SPLINE
SPL {X  -129.366, Y  +765.635, Z    +0.000, E1   +44.361, E3 -207865.968}
SPL {X  -144.719, Y  +739.715, Z    +0.000, E1   +37.620, E3 -207892.815}
SPL {X  -154.606, Y  +712.654, Z    +0.000, E1   +26.872, E3 -207906.035}
SPL {X  -158.229, Y  +695.175, Z    +0.000, E1   +17.621, E3 -207910.521}
SPL {X  -159.735, Y  +680.532, Z    +0.000, E1    +8.352, E3 -207912.613}
SPL {X  -159.976, Y  +673.579, Z    +0.000, E1    +3.308, E3 -207913.108}
SPL {X  -159.990, Y  +669.438, Z    +0.000, E1    +0.061, E3 -207913.205}
SPL {X  -159.990, Y  +667.221, Z    +0.000, E1    -2.789, E3 -207913.248}
SPL {X  -159.990, Y  +663.611, Z    +0.000, E1    -7.967, E3 -207913.439}
SPL {X  -159.990, Y  +658.381, Z    +0.000, E1   -16.786, E3 -207913.919}
SPL {X  -159.990, Y  +651.878, Z    +0.000, E1   -27.298, E3 -207914.918}
SPL {X  -159.990, Y  +644.587, Z    +0.000, E1   -37.284, E3 -207916.501}
SPL {X  -159.990, Y  +633.621, Z    +0.000, E1   -47.309, E3 -207919.992}
SPL {X  -159.990, Y  +588.658, Z    +0.000, E1   -60.812, E3 -207942.312}
SPL {X  -159.990, Y  +495.038, Z    +0.000, E1   -63.580, E3 -208017.548}
SPL {X  -159.990, Y  +483.848, Z    +0.000, E1   -63.590, E3 -208029.333}
SPL {X  -159.990, Y  +471.874, Z    +0.000, E1   -63.586, E3 -208041.959}
SPL {X  -159.990, Y  +461.079, Z    +0.000, E1   -63.579, E3 -208053.367}
SPL {X  -159.990, Y  +450.188, Z    +0.000, E1   -63.581, E3 -208064.858}
SPL {X  -159.990, Y  +442.553, Z    +0.000, E1   -63.337, E3 -208074.682}
ENDSPLINE

SPLINE
SPL {X  -159.990, Y  +465.419, Z    +0.000, E1   -58.181, E3 -208083.527}
ENDSPLINE

SPLINE
SPL {X  -159.990, Y  +455.003, Z    +0.000, E1   -58.788, E3 -208093.065}
SPL {X  -159.990, Y  +443.180, Z    +0.000, E1   -59.522, E3 -208103.103}
SPL {X  -159.990, Y  +431.227, Z    +0.000, E1   -60.120, E3 -208113.796}
SPL {X  -159.990, Y  +413.464, Z    +0.000, E1   -61.043, E3 -208128.786}
SPL {X  -159.990, Y  +395.417, Z    +0.000, E1   -62.063, E3 -208142.228}
SPL {X  -159.983, Y  +381.042, Z    +0.000, E1   -62.802, E3 -208152.860}
SPL {X  -159.542, Y  +370.537, Z    +0.000, E1   -63.069, E3 -208162.242}
SPL {X  -158.758, Y  +362.683, Z    +0.000, E1   -62.956, E3 -208171.515}
SPL {X  -157.125, Y  +352.357, Z    +0.000, E1   -62.751, E3 -208184.249}
SPL {X  -154.421, Y  +340.656, Z    +0.000, E1   -62.344, E3 -208199.602}
SPL {X  -151.938, Y  +332.383, Z    +0.000, E1   -61.927, E3 -208211.075}
SPL {X  -149.604, Y  +325.796, Z    +0.000, E1   -61.568, E3 -208220.461}
SPL {X  -147.413, Y  +320.320, Z    +0.000, E1   -61.198, E3 -208228.514}
SPL {X  -145.235, Y  +315.391, Z    +0.000, E1   -60.847, E3 -208235.888}
SPL {X  -141.610, Y  +308.046, Z    +0.000, E1   -60.266, E3 -208247.125}
SPL {X  -138.010, Y  +301.568, Z    +0.000, E1   -59.585, E3 -208257.396}
SPL {X  -134.495, Y  +295.853, Z    +0.000, E1   -58.965, E3 -208266.533}
SPL {X  -113.541, Y  +269.782, Z    +0.000, E1   -50.113, E3 -208374.126}
ENDSPLINE

SPLINE
SPL {X  -141.985, Y  +308.763, Z    +0.000, E1   -38.695, E3 -208482.078}
SPL {X  -154.491, Y  +340.913, Z    +0.000, E1   -26.570, E3 -208500.531}
SPL {X  -158.582, Y  +361.322, Z    +0.000, E1   -15.773, E3 -208506.129}
SPL {X  -159.657, Y  +372.183, Z    +0.000, E1    -8.995, E3 -208507.738}
SPL {X  -159.949, Y  +378.873, Z    +0.000, E1    -4.398, E3 -208508.312}
SPL {X  -159.990, Y  +384.063, Z    +0.000, E1    -0.515, E3 -208508.508}
SPL {X  -159.990, Y  +386.497, Z    +0.000, E1    +2.123, E3 -208508.564}
SPL {X  -159.990, Y  +389.673, Z    +0.000, E1    +6.604, E3 -208508.717}
SPL {X  -159.990, Y  +394.848, Z    +0.000, E1   +14.441, E3 -208509.206}
SPL {X  -159.990, Y  +402.771, Z    +0.000, E1   +27.045, E3 -208510.458}
SPL {X  -159.990, Y  +414.719, Z    +0.000, E1   +41.161, E3 -208513.632}
SPL {X  -159.990, Y  +424.336, Z    +0.000, E1   +48.481, E3 -208517.066}
SPL {X  -159.990, Y  +469.763, Z    +0.000, E1   +60.937, E3 -208539.355}
SPL {X  -159.990, Y  +561.242, Z    +0.000, E1   +63.988, E3 -208610.303}
SPL {X  -159.990, Y  +574.019, Z    +0.000, E1   +64.020, E3 -208623.469}
SPL {X  -159.990, Y  +588.139, Z    +0.000, E1   +64.000, E3 -208638.117}
SPL {X  -159.990, Y  +601.786, Z    +0.000, E1   +64.016, E3 -208652.221}
SPL {X  -159.990, Y  +614.683, Z    +0.000, E1   +63.997, E3 -208665.590}
SPL {X  -159.990, Y  +629.274, Z    +0.000, E1   +64.033, E3 -208680.621}
SPL {X  -159.990, Y  +645.396, Z    +0.000, E1   +64.010, E3 -208697.352}
SPL {X  -159.990, Y  +656.294, Z    +0.000, E1   +63.988, E3 -208708.681}
SPL {X  -159.990, Y  +667.666, Z    +0.000, E1   +64.016, E3 -208720.373}
SPL {X  -159.767, Y  +679.937, Z    +0.000, E1   +63.968, E3 -208733.348}
SPL {X  -158.736, Y  +691.491, Z    +0.000, E1   +63.843, E3 -208746.347}
SPL {X  -157.131, Y  +701.612, Z    +0.000, E1   +63.591, E3 -208758.537}
SPL {X  -154.918, Y  +711.464, Z    +0.000, E1   +63.294, E3 -208770.972}
SPL {X  -152.656, Y  +719.385, Z    +0.000, E1   +62.921, E3 -208781.540}
SPL {X  -150.233, Y  +726.516, Z    +0.000, E1   +62.565, E3 -208791.318}
SPL {X  -147.385, Y  +733.745, Z    +0.000, E1   +62.104, E3 -208801.623}
SPL {X  -144.667, Y  +739.825, Z    +0.000, E1   +61.658, E3 -208810.525}
SPL {X  -142.263, Y  +744.698, Z    +0.000, E1   +61.245, E3 -208817.840}
SPL {X  -138.935, Y  +750.833, Z    +0.000, E1   +60.711, E3 -208827.165}
SPL {X  -135.668, Y  +756.300, Z    +0.000, E1   +60.086, E3 -208835.728}
SPL {X  -132.995, Y  +760.433, Z    +0.000, E1   +59.601, E3 -208842.235}
SPL {X  -109.949, Y  +787.724, Z    +0.000, E1   +51.944, E3 -208934.797}
ENDSPLINE

SPLINE
SPL {X  -129.366, Y  +765.635, Z    +0.000, E1   +44.361, E3 -209044.539}
SPL {X  -144.719, Y  +739.715, Z    +0.000, E1   +37.620, E3 -209071.386}
SPL {X  -154.606, Y  +712.654, Z    +0.000, E1   +26.872, E3 -209084.606}
SPL {X  -158.229, Y  +695.175, Z    +0.000, E1   +17.621, E3 -209089.092}
SPL {X  -159.735, Y  +680.532, Z    +0.000, E1    +8.352, E3 -209091.185}
SPL {X  -159.976, Y  +673.579, Z    +0.000, E1    +3.308, E3 -209091.679}
SPL {X  -159.990, Y  +669.438, Z    +0.000, E1    +0.061, E3 -209091.777}
SPL {X  -159.990, Y  +666.135, Z    +0.000, E1    -4.178, E3 -209091.868}
SPL {X  -159.990, Y  +662.249, Z    +0.000, E1   -10.338, E3 -209092.099}
SPL {X  -159.990, Y  +658.381, Z    +0.000, E1   -16.786, E3 -209092.491}
SPL {X  -159.990, Y  +651.878, Z    +0.000, E1   -27.298, E3 -209093.490}
SPL {X  -159.990, Y  +644.587, Z    +0.000, E1   -37.284, E3 -209095.073}
SPL {X  -159.990, Y  +633.621, Z    +0.000, E1   -47.309, E3 -209098.564}
SPL {X  -159.990, Y  +588.658, Z    +0.000, E1   -60.812, E3 -209120.884}
SPL {X  -159.990, Y  +495.038, Z    +0.000, E1   -63.580, E3 -209196.120}
SPL {X  -159.990, Y  +483.848, Z    +0.000, E1   -63.590, E3 -209207.905}
SPL {X  -159.990, Y  +471.874, Z    +0.000, E1   -63.586, E3 -209220.530}
SPL {X  -159.990, Y  +461.079, Z    +0.000, E1   -63.579, E3 -209231.939}
SPL {X  -159.990, Y  +450.188, Z    +0.000, E1   -63.581, E3 -209243.429}
SPL {X  -159.990, Y  +442.553, Z    +0.000, E1   -63.337, E3 -209253.253}
ENDSPLINE

SPLINE
SPL {X  -159.990, Y  +465.419, Z    +0.000, E1   -58.181, E3 -209262.098}
ENDSPLINE

SPLINE
SPL {X  -159.990, Y  +455.003, Z    +0.000, E1   -58.788, E3 -209271.637}
SPL {X  -159.990, Y  +443.180, Z    +0.000, E1   -59.522, E3 -209281.675}
SPL {X  -159.990, Y  +431.227, Z    +0.000, E1   -60.120, E3 -209292.367}
SPL {X  -159.990, Y  +413.464, Z    +0.000, E1   -61.043, E3 -209307.357}
SPL {X  -159.990, Y  +395.417, Z    +0.000, E1   -62.063, E3 -209320.800}
SPL {X  -159.983, Y  +381.042, Z    +0.000, E1   -62.802, E3 -209331.431}
SPL {X  -159.542, Y  +370.537, Z    +0.000, E1   -63.069, E3 -209340.813}
SPL {X  -158.287, Y  +359.218, Z    +0.000, E1   -62.927, E3 -209354.228}
SPL {X  -156.553, Y  +349.515, Z    +0.000, E1   -62.627, E3 -209366.539}
SPL {X  -154.421, Y  +340.656, Z    +0.000, E1   -62.344, E3 -209378.173}
SPL {X  -151.938, Y  +332.383, Z    +0.000, E1   -61.927, E3 -209389.646}
SPL {X  -149.604, Y  +325.796, Z    +0.000, E1   -61.568, E3 -209399.032}
SPL {X  -147.413, Y  +320.320, Z    +0.000, E1   -61.198, E3 -209407.085}
SPL {X  -145.235, Y  +315.391, Z    +0.000, E1   -60.847, E3 -209414.460}
SPL {X  -141.610, Y  +308.046, Z    +0.000, E1   -60.266, E3 -209425.696}
SPL {X  -138.010, Y  +301.568, Z    +0.000, E1   -59.585, E3 -209435.967}
SPL {X  -134.495, Y  +295.853, Z    +0.000, E1   -58.965, E3 -209445.105}
SPL {X  -113.541, Y  +269.782, Z    +0.000, E1   -50.113, E3 -209552.697}
ENDSPLINE

SPLINE
SPL {X  -141.985, Y  +308.763, Z    +0.000, E1   -38.695, E3 -209660.650}
SPL {X  -154.491, Y  +340.913, Z    +0.000, E1   -26.570, E3 -209679.102}
SPL {X  -158.582, Y  +361.322, Z    +0.000, E1   -15.773, E3 -209684.701}
SPL {X  -159.657, Y  +372.183, Z    +0.000, E1    -8.995, E3 -209686.309}
SPL {X  -159.949, Y  +378.873, Z    +0.000, E1    -4.398, E3 -209686.883}
SPL {X  -159.990, Y  +384.063, Z    +0.000, E1    -0.515, E3 -209687.079}
SPL {X  -159.990, Y  +386.497, Z    +0.000, E1    +2.123, E3 -209687.135}
SPL {X  -159.990, Y  +391.572, Z    +0.000, E1    +9.236, E3 -209687.441}
SPL {X  -159.990, Y  +397.198, Z    +0.000, E1   +18.490, E3 -209688.066}
SPL {X  -159.990, Y  +402.771, Z    +0.000, E1   +27.045, E3 -209689.029}
SPL {X  -159.990, Y  +416.096, Z    +0.000, E1   +42.325, E3 -209692.696}
SPL {X  -159.990, Y  +469.763, Z    +0.000, E1   +60.937, E3 -209717.926}
SPL {X  -159.990, Y  +565.969, Z    +0.000, E1   +64.023, E3 -209793.700}
SPL {X  -159.990, Y  +578.082, Z    +0.000, E1   +63.987, E3 -209806.309}
SPL {X  -159.990, Y  +588.139, Z    +0.000, E1   +64.000, E3 -209816.689}
SPL {X  -159.990, Y  +601.786, Z    +0.000, E1   +64.016, E3 -209830.793}
SPL {X  -159.990, Y  +618.770, Z    +0.000, E1   +64.031, E3 -209848.329}
SPL {X  -159.990, Y  +636.111, Z    +0.000, E1   +64.024, E3 -209866.284}
SPL {X  -159.990, Y  +652.385, Z    +0.000, E1   +64.020, E3 -209883.141}
SPL {X  -159.990, Y  +667.666, Z    +0.000, E1   +64.016, E3 -209898.945}
SPL {X  -159.767, Y  +679.937, Z    +0.000, E1   +63.968, E3 -209911.920}
SPL {X  -159.113, Y  +688.225, Z    +0.000, E1   +63.867, E3 -209921.198}
SPL {X  -158.361, Y  +694.273, Z    +0.000, E1   +63.762, E3 -209928.235}
SPL {X  -157.131, Y  +701.612, Z    +0.000, E1   +63.591, E3 -209937.108}
SPL {X  -154.918, Y  +711.464, Z    +0.000, E1   +63.294, E3 -209949.543}
SPL {X  -151.874, Y  +721.810, Z    +0.000, E1   +62.834, E3 -209963.350}
SPL {X  -148.087, Y  +732.056, Z    +0.000, E1   +62.252, E3 -209977.707}
SPL {X  -144.667, Y  +739.825, Z    +0.000, E1   +61.658, E3 -209989.096}
SPL {X  -142.263, Y  +744.698, Z    +0.000, E1   +61.245, E3 -209996.412}
SPL {X  -138.935, Y  +750.833, Z    +0.000, E1   +60.711, E3 -210005.736}
SPL {X  -135.668, Y  +756.300, Z    +0.000, E1   +60.086, E3 -210014.299}
SPL {X  -132.995, Y  +760.433, Z    +0.000, E1   +59.601, E3 -210020.807}
SPL {X  -109.949, Y  +787.724, Z    +0.000, E1   +51.944, E3 -210113.368}
ENDSPLINE

SPLINE
SPL {X  -129.366, Y  +765.635, Z    +0.000, E1   +44.361, E3 -210223.110}
SPL {X  -144.719, Y  +739.715, Z    +0.000, E1   +37.620, E3 -210249.958}
SPL {X  -154.606, Y  +712.654, Z    +0.000, E1   +26.872, E3 -210263.178}
SPL {X  -158.229, Y  +695.175, Z    +0.000, E1   +17.621, E3 -210267.664}
SPL {X  -159.536, Y  +683.548, Z    +0.000, E1   +10.326, E3 -210269.452}
SPL {X  -159.946, Y  +675.243, Z    +0.000, E1    +4.608, E3 -210270.160}
SPL {X  -159.990, Y  +669.438, Z    +0.000, E1    +0.061, E3 -210270.348}
SPL {X  -159.990, Y  +666.135, Z    +0.000, E1    -4.178, E3 -210270.439}
SPL {X  -159.990, Y  +662.249, Z    +0.000, E1   -10.338, E3 -210270.671}
SPL {X  -159.990, Y  +658.381, Z    +0.000, E1   -16.786, E3 -210271.062}
SPL {X  -159.990, Y  +651.878, Z    +0.000, E1   -27.298, E3 -210272.061}
SPL {X  -159.990, Y  +644.587, Z    +0.000, E1   -37.284, E3 -210273.644}
SPL {X  -159.990, Y  +633.621, Z    +0.000, E1   -47.309, E3 -210277.135}
SPL {X  -159.990, Y  +588.658, Z    +0.000, E1   -60.812, E3 -210299.455}
SPL {X  -159.990, Y  +495.038, Z    +0.000, E1   -63.580, E3 -210374.691}
SPL {X  -159.990, Y  +483.848, Z    +0.000, E1   -63.590, E3 -210386.476}
SPL {X  -159.990, Y  +471.874, Z    +0.000, E1   -63.586, E3 -210399.102}
SPL {X  -159.990, Y  +461.079, Z    +0.000, E1   -63.579, E3 -210410.510}
SPL {X  -159.990, Y  +450.188, Z    +0.000, E1   -63.581, E3 -210422.001}
SPL {X  -159.990, Y  +442.553, Z    +0.000, E1   -63.337, E3 -210431.824}
ENDSPLINE

SPLINE
SPL {X  -159.990, Y  +465.419, Z    +0.000, E1   -58.181, E3 -210440.670}
ENDSPLINE

SPLINE
SPL {X  -159.990, Y  +455.003, Z    +0.000, E1   -58.788, E3 -210450.208}
SPL {X  -159.990, Y  +443.180, Z    +0.000, E1   -59.522, E3 -210460.246}
SPL {X  -159.990, Y  +431.227, Z    +0.000, E1   -60.120, E3 -210470.938}
SPL {X  -159.990, Y  +413.464, Z    +0.000, E1   -61.043, E3 -210485.928}
SPL {X  -159.990, Y  +395.417, Z    +0.000, E1   -62.063, E3 -210499.371}
SPL {X  -159.983, Y  +381.042, Z    +0.000, E1   -62.802, E3 -210510.003}
SPL {X  -159.542, Y  +370.537, Z    +0.000, E1   -63.069, E3 -210519.385}
SPL {X  -158.758, Y  +362.683, Z    +0.000, E1   -62.956, E3 -210528.658}
SPL {X  -157.125, Y  +352.357, Z    +0.000, E1   -62.751, E3 -210541.392}
SPL {X  -154.421, Y  +340.656, Z    +0.000, E1   -62.344, E3 -210556.745}
SPL {X  -151.938, Y  +332.383, Z    +0.000, E1   -61.927, E3 -210568.218}
SPL {X  -149.604, Y  +325.796, Z    +0.000, E1   -61.568, E3 -210577.603}
SPL {X  -147.413, Y  +320.320, Z    +0.000, E1   -61.198, E3 -210585.657}
SPL {X  -145.235, Y  +315.391, Z    +0.000, E1   -60.847, E3 -210593.031}
SPL {X  -141.610, Y  +308.046, Z    +0.000, E1   -60.266, E3 -210604.268}
SPL {X  -138.010, Y  +301.568, Z    +0.000, E1   -59.585, E3 -210614.539}
SPL {X  -134.495, Y  +295.853, Z    +0.000, E1   -58.965, E3 -210623.676}
SPL {X  -113.541, Y  +269.782, Z    +0.000, E1   -50.113, E3 -210731.269}
ENDSPLINE

SPLINE
SPL {X  -141.985, Y  +308.763, Z    +0.000, E1   -38.695, E3 -210839.221}
SPL {X  -154.491, Y  +340.913, Z    +0.000, E1   -26.570, E3 -210857.674}
SPL {X  -158.582, Y  +361.322, Z    +0.000, E1   -15.773, E3 -210863.272}
SPL {X  -159.657, Y  +372.183, Z    +0.000, E1    -8.995, E3 -210864.880}
SPL {X  -159.949, Y  +378.873, Z    +0.000, E1    -4.398, E3 -210865.455}
SPL {X  -159.990, Y  +384.063, Z    +0.000, E1    -0.515, E3 -210865.651}
SPL {X  -159.990, Y  +386.497, Z    +0.000, E1    +2.123, E3 -210865.707}
SPL {X  -159.990, Y  +391.572, Z    +0.000, E1    +9.236, E3 -210866.013}
SPL {X  -159.990, Y  +397.198, Z    +0.000, E1   +18.490, E3 -210866.637}
SPL {X  -159.990, Y  +402.771, Z    +0.000, E1   +27.045, E3 -210867.601}
SPL {X  -159.990, Y  +416.096, Z    +0.000, E1   +42.325, E3 -210871.268}
SPL {X  -159.990, Y  +469.763, Z    +0.000, E1   +60.937, E3 -210896.498}
SPL {X  -159.990, Y  +565.969, Z    +0.000, E1   +64.023, E3 -210972.272}
SPL {X  -159.990, Y  +578.082, Z    +0.000, E1   +63.987, E3 -210984.880}
SPL {X  -159.990, Y  +588.139, Z    +0.000, E1   +64.000, E3 -210995.260}
SPL {X  -159.990, Y  +601.786, Z    +0.000, E1   +64.016, E3 -211009.364}
SPL {X  -159.990, Y  +618.770, Z    +0.000, E1   +64.031, E3 -211026.900}
SPL {X  -159.990, Y  +632.928, Z    +0.000, E1   +63.998, E3 -211041.609}
SPL {X  -159.990, Y  +645.396, Z    +0.000, E1   +64.010, E3 -211054.495}
SPL {X  -159.990, Y  +659.675, Z    +0.000, E1   +64.013, E3 -211069.267}
SPL {X  -159.990, Y  +670.719, Z    +0.000, E1   +63.993, E3 -211080.716}
SPL {X  -159.767, Y  +679.937, Z    +0.000, E1   +63.968, E3 -211090.491}
SPL {X  -158.736, Y  +691.491, Z    +0.000, E1   +63.843, E3 -211103.490}
SPL {X  -157.131, Y  +701.612, Z    +0.000, E1   +63.591, E3 -211115.680}
SPL {X  -155.594, Y  +708.746, Z    +0.000, E1   +63.361, E3 -211124.660}
SPL {X  -153.286, Y  +717.329, Z    +0.000, E1   +63.046, E3 -211135.868}
SPL {X  -150.953, Y  +724.510, Z    +0.000, E1   +62.654, E3 -211145.696}
SPL {X  -148.087, Y  +732.056, Z    +0.000, E1   +62.252, E3 -211156.278}
SPL {X  -144.667, Y  +739.825, Z    +0.000, E1   +61.658, E3 -211167.668}
SPL {X  -142.263, Y  +744.698, Z    +0.000, E1   +61.245, E3 -211174.983}
SPL {X  -139.956, Y  +749.019, Z    +0.000, E1   +60.852, E3 -211181.560}
SPL {X  -136.617, Y  +754.762, Z    +0.000, E1   +60.296, E3 -211190.415}
SPL {X  -132.995, Y  +760.433, Z    +0.000, E1   +59.601, E3 -211199.378}
SPL {X  -109.949, Y  +787.724, Z    +0.000, E1   +51.944, E3 -211291.940}
ENDSPLINE

SPLINE
SPL {X  -129.366, Y  +765.635, Z    +0.000, E1   +44.361, E3 -211401.682}
SPL {X  -144.719, Y  +739.715, Z    +0.000, E1   +37.620, E3 -211428.529}
SPL {X  -154.606, Y  +712.654, Z    +0.000, E1   +26.872, E3 -211441.749}
SPL {X  -158.229, Y  +695.175, Z    +0.000, E1   +17.621, E3 -211446.235}
SPL {X  -159.536, Y  +683.548, Z    +0.000, E1   +10.326, E3 -211448.023}
SPL {X  -159.946, Y  +675.243, Z    +0.000, E1    +4.608, E3 -211448.732}
SPL {X  -159.990, Y  +669.438, Z    +0.000, E1    +0.061, E3 -211448.919}
SPL {X  -159.990, Y  +666.135, Z    +0.000, E1    -4.178, E3 -211449.011}
SPL {X  -159.990, Y  +662.249, Z    +0.000, E1   -10.338, E3 -211449.242}
SPL {X  -159.990, Y  +658.381, Z    +0.000, E1   -16.786, E3 -211449.634}
SPL {X  -159.990, Y  +651.878, Z    +0.000, E1   -27.298, E3 -211450.633}
SPL {X  -159.990, Y  +644.587, Z    +0.000, E1   -37.284, E3 -211452.216}
SPL {X  -159.990, Y  +633.621, Z    +0.000, E1   -47.309, E3 -211455.707}
SPL {X  -159.990, Y  +588.658, Z    +0.000, E1   -60.812, E3 -211478.026}
SPL {X  -159.990, Y  +495.038, Z    +0.000, E1   -63.580, E3 -211553.263}
SPL {X  -159.990, Y  +483.848, Z    +0.000, E1   -63.590, E3 -211565.047}
SPL {X  -159.990, Y  +471.874, Z    +0.000, E1   -63.586, E3 -211577.673}
SPL {X  -159.990, Y  +461.079, Z    +0.000, E1   -63.579, E3 -211589.082}
SPL {X  -159.990, Y  +450.188, Z    +0.000, E1   -63.581, E3 -211600.572}
SPL {X  -159.990, Y  +442.553, Z    +0.000, E1   -63.337, E3 -211610.396}
ENDSPLINE

SPLINE
SPL {X  -159.990, Y  +465.419, Z    +0.000, E1   -58.181, E3 -211619.241}
ENDSPLINE

SPLINE
SPL {X  -159.990, Y  +455.003, Z    +0.000, E1   -58.788, E3 -211628.779}
SPL {X  -159.990, Y  +443.180, Z    +0.000, E1   -59.522, E3 -211638.818}
SPL {X  -159.990, Y  +431.227, Z    +0.000, E1   -60.120, E3 -211649.510}
SPL {X  -159.990, Y  +413.464, Z    +0.000, E1   -61.043, E3 -211664.500}
SPL {X  -159.990, Y  +395.417, Z    +0.000, E1   -62.063, E3 -211677.943}
SPL {X  -159.983, Y  +381.042, Z    +0.000, E1   -62.802, E3 -211688.574}
SPL {X  -159.542, Y  +370.537, Z    +0.000, E1   -63.069, E3 -211697.956}
SPL {X  -158.758, Y  +362.683, Z    +0.000, E1   -62.956, E3 -211707.230}
SPL {X  -157.125, Y  +352.357, Z    +0.000, E1   -62.751, E3 -211719.963}
SPL {X  -154.421, Y  +340.656, Z    +0.000, E1   -62.344, E3 -211735.316}
SPL {X  -151.938, Y  +332.383, Z    +0.000, E1   -61.927, E3 -211746.789}
SPL {X  -149.604, Y  +325.796, Z    +0.000, E1   -61.568, E3 -211756.175}
SPL {X  -147.413, Y  +320.320, Z    +0.000, E1   -61.198, E3 -211764.228}
SPL {X  -145.235, Y  +315.391, Z    +0.000, E1   -60.847, E3 -211771.603}
SPL {X  -141.610, Y  +308.046, Z    +0.000, E1   -60.266, E3 -211782.839}
SPL {X  -138.010, Y  +301.568, Z    +0.000, E1   -59.585, E3 -211793.110}
SPL {X  -134.495, Y  +295.853, Z    +0.000, E1   -58.965, E3 -211802.248}
SPL {X  -113.541, Y  +269.782, Z    +0.000, E1   -50.113, E3 -211909.840}
ENDSPLINE

SPLINE
SPL {X  -141.985, Y  +308.763, Z    +0.000, E1   -38.695, E3 -212017.793}
SPL {X  -154.491, Y  +340.913, Z    +0.000, E1   -26.570, E3 -212036.245}
SPL {X  -158.582, Y  +361.322, Z    +0.000, E1   -15.773, E3 -212041.844}
SPL {X  -159.657, Y  +372.183, Z    +0.000, E1    -8.995, E3 -212043.452}
SPL {X  -159.949, Y  +378.873, Z    +0.000, E1    -4.398, E3 -212044.026}
SPL {X  -159.990, Y  +384.063, Z    +0.000, E1    -0.515, E3 -212044.222}
SPL {X  -159.990, Y  +386.497, Z    +0.000, E1    +2.123, E3 -212044.278}
SPL {X  -159.990, Y  +389.673, Z    +0.000, E1    +6.604, E3 -212044.431}
SPL {X  -159.990, Y  +394.848, Z    +0.000, E1   +14.441, E3 -212044.920}
SPL {X  -159.990, Y  +402.771, Z    +0.000, E1   +27.045, E3 -212046.172}
SPL {X  -159.990, Y  +414.719, Z    +0.000, E1   +41.161, E3 -212049.346}
SPL {X  -159.990, Y  +424.336, Z    +0.000, E1   +48.481, E3 -212052.781}
SPL {X  -159.990, Y  +469.763, Z    +0.000, E1   +60.937, E3 -212075.069}
SPL {X  -159.990, Y  +561.242, Z    +0.000, E1   +63.988, E3 -212146.017}
SPL {X  -159.990, Y  +574.019, Z    +0.000, E1   +64.020, E3 -212159.184}
SPL {X  -159.990, Y  +588.139, Z    +0.000, E1   +64.000, E3 -212173.832}
SPL {X  -159.990, Y  +601.786, Z    +0.000, E1   +64.016, E3 -212187.935}
SPL {X  -159.990, Y  +614.683, Z    +0.000, E1   +63.997, E3 -212201.304}
SPL {X  -159.990, Y  +629.274, Z    +0.000, E1   +64.033, E3 -212216.335}
SPL {X  -159.990, Y  +645.396, Z    +0.000, E1   +64.010, E3 -212233.066}
SPL {X  -159.990, Y  +656.294, Z    +0.000, E1   +63.988, E3 -212244.396}
SPL {X  -159.990, Y  +667.666, Z    +0.000, E1   +64.016, E3 -212256.087}
SPL {X  -159.767, Y  +679.937, Z    +0.000, E1   +63.968, E3 -212269.063}
SPL {X  -158.736, Y  +691.491, Z    +0.000, E1   +63.843, E3 -212282.061}
SPL {X  -157.131, Y  +701.612, Z    +0.000, E1   +63.591, E3 -212294.251}
SPL {X  -154.918, Y  +711.464, Z    +0.000, E1   +63.294, E3 -212306.686}
SPL {X  -152.656, Y  +719.385, Z    +0.000, E1   +62.921, E3 -212317.255}
SPL {X  -150.233, Y  +726.516, Z    +0.000, E1   +62.565, E3 -212327.033}
SPL {X  -147.385, Y  +733.745, Z    +0.000, E1   +62.104, E3 -212337.337}
SPL {X  -144.667, Y  +739.825, Z    +0.000, E1   +61.658, E3 -212346.239}
SPL {X  -142.263, Y  +744.698, Z    +0.000, E1   +61.245, E3 -212353.554}
SPL {X  -138.935, Y  +750.833, Z    +0.000, E1   +60.711, E3 -212362.879}
SPL {X  -135.668, Y  +756.300, Z    +0.000, E1   +60.086, E3 -212371.442}
SPL {X  -132.995, Y  +760.433, Z    +0.000, E1   +59.601, E3 -212377.950}
SPL {X  -109.949, Y  +787.724, Z    +0.000, E1   +51.944, E3 -212470.511}
ENDSPLINE

SPLINE
SPL {X  -129.366, Y  +765.635, Z    +0.000, E1   +44.361, E3 -212580.253}
SPL {X  -144.719, Y  +739.715, Z    +0.000, E1   +37.620, E3 -212607.101}
SPL {X  -154.606, Y  +712.654, Z    +0.000, E1   +26.872, E3 -212620.321}
SPL {X  -158.229, Y  +695.175, Z    +0.000, E1   +17.621, E3 -212624.807}
SPL {X  -159.735, Y  +680.532, Z    +0.000, E1    +8.352, E3 -212626.899}
SPL {X  -159.976, Y  +673.579, Z    +0.000, E1    +3.308, E3 -212627.393}
SPL {X  -159.990, Y  +669.438, Z    +0.000, E1    +0.061, E3 -212627.491}
SPL {X  -159.990, Y  +666.135, Z    +0.000, E1    -4.178, E3 -212627.582}
SPL {X  -159.990, Y  +662.249, Z    +0.000, E1   -10.338, E3 -212627.813}
SPL {X  -159.990, Y  +658.381, Z    +0.000, E1   -16.786, E3 -212628.205}
SPL {X  -159.990, Y  +651.878, Z    +0.000, E1   -27.298, E3 -212629.204}
SPL {X  -159.990, Y  +644.587, Z    +0.000, E1   -37.284, E3 -212630.787}
SPL {X  -159.990, Y  +633.621, Z    +0.000, E1   -47.309, E3 -212634.278}
SPL {X  -159.990, Y  +588.658, Z    +0.000, E1   -60.812, E3 -212656.598}
SPL {X  -159.990, Y  +495.038, Z    +0.000, E1   -63.580, E3 -212731.834}
SPL {X  -159.990, Y  +483.848, Z    +0.000, E1   -63.590, E3 -212743.619}
SPL {X  -159.990, Y  +471.874, Z    +0.000, E1   -63.586, E3 -212756.245}
SPL {X  -159.990, Y  +461.079, Z    +0.000, E1   -63.579, E3 -212767.653}
SPL {X  -159.990, Y  +450.188, Z    +0.000, E1   -63.581, E3 -212779.144}
SPL {X  -159.990, Y  +442.553, Z    +0.000, E1   -63.337, E3 -212788.967}
ENDSPLINE

SPLINE
SPL {X  -159.990, Y  +465.419, Z    +0.000, E1   -58.181, E3 -212797.813}
ENDSPLINE

SPLINE
SPL {X  -159.990, Y  +455.003, Z    +0.000, E1   -58.788, E3 -212807.351}
SPL {X  -159.990, Y  +443.180, Z    +0.000, E1   -59.522, E3 -212817.389}
SPL {X  -159.990, Y  +431.227, Z    +0.000, E1   -60.120, E3 -212828.081}
SPL {X  -159.990, Y  +413.464, Z    +0.000, E1   -61.043, E3 -212843.071}
SPL {X  -159.990, Y  +395.417, Z    +0.000, E1   -62.063, E3 -212856.514}
SPL {X  -159.983, Y  +381.042, Z    +0.000, E1   -62.802, E3 -212867.145}
SPL {X  -159.542, Y  +370.537, Z    +0.000, E1   -63.069, E3 -212876.527}
SPL {X  -158.287, Y  +359.218, Z    +0.000, E1   -62.927, E3 -212889.942}
SPL {X  -156.553, Y  +349.515, Z    +0.000, E1   -62.627, E3 -212902.254}
SPL {X  -154.421, Y  +340.656, Z    +0.000, E1   -62.344, E3 -212913.888}
SPL {X  -151.938, Y  +332.383, Z    +0.000, E1   -61.927, E3 -212925.360}
SPL {X  -149.604, Y  +325.796, Z    +0.000, E1   -61.568, E3 -212934.746}
SPL {X  -147.413, Y  +320.320, Z    +0.000, E1   -61.198, E3 -212942.799}
SPL {X  -145.235, Y  +315.391, Z    +0.000, E1   -60.847, E3 -212950.174}
SPL {X  -141.610, Y  +308.046, Z    +0.000, E1   -60.266, E3 -212961.410}
SPL {X  -138.010, Y  +301.568, Z    +0.000, E1   -59.585, E3 -212971.682}
SPL {X  -134.495, Y  +295.853, Z    +0.000, E1   -58.965, E3 -212980.819}
SPL {X  -113.541, Y  +269.782, Z    +0.000, E1   -50.113, E3 -213088.412}
ENDSPLINE

SPLINE
SPL {X  -141.985, Y  +308.763, Z    +0.000, E1   -38.695, E3 -213196.364}
SPL {X  -154.491, Y  +340.913, Z    +0.000, E1   -26.570, E3 -213214.816}
SPL {X  -158.582, Y  +361.322, Z    +0.000, E1   -15.773, E3 -213220.415}
SPL {X  -159.657, Y  +372.183, Z    +0.000, E1    -8.995, E3 -213222.023}
SPL {X  -159.949, Y  +378.873, Z    +0.000, E1    -4.398, E3 -213222.598}
SPL {X  -159.990, Y  +384.063, Z    +0.000, E1    -0.515, E3 -213222.794}
SPL {X  -159.990, Y  +386.497, Z    +0.000, E1    +2.123, E3 -213222.850}
SPL {X  -159.990, Y  +391.572, Z    +0.000, E1    +9.236, E3 -213223.156}
SPL {X  -159.990, Y  +397.198, Z    +0.000, E1   +18.490, E3 -213223.780}
SPL {X  -159.990, Y  +402.771, Z    +0.000, E1   +27.045, E3 -213224.743}
SPL {X  -159.990, Y  +416.096, Z    +0.000, E1   +42.325, E3 -213228.411}
SPL {X  -159.990, Y  +469.763, Z    +0.000, E1   +60.937, E3 -213253.641}
SPL {X  -159.990, Y  +565.969, Z    +0.000, E1   +64.023, E3 -213329.414}
SPL {X  -159.990, Y  +578.082, Z    +0.000, E1   +63.987, E3 -213342.023}
SPL {X  -159.990, Y  +588.139, Z    +0.000, E1   +64.000, E3 -213352.403}
SPL {X  -159.990, Y  +601.786, Z    +0.000, E1   +64.016, E3 -213366.507}
SPL {X  -159.990, Y  +618.770, Z    +0.000, E1   +64.031, E3 -213384.043}
SPL {X  -159.990, Y  +636.111, Z    +0.000, E1   +64.024, E3 -213401.998}
SPL {X  -159.990, Y  +652.385, Z    +0.000, E1   +64.020, E3 -213418.855}
SPL {X  -159.990, Y  +667.666, Z    +0.000, E1   +64.016, E3 -213434.659}
SPL {X  -159.767, Y  +679.937, Z    +0.000, E1   +63.968, E3 -213447.634}
SPL {X  -159.113, Y  +688.225, Z    +0.000, E1   +63.867, E3 -213456.912}
SPL {X  -158.361, Y  +694.273, Z    +0.000, E1   +63.762, E3 -213463.950}
SPL {X  -157.131, Y  +701.612, Z    +0.000, E1   +63.591, E3 -213472.823}
SPL {X  -155.594, Y  +708.746, Z    +0.000, E1   +63.361, E3 -213481.803}
SPL {X  -153.286, Y  +717.329, Z    +0.000, E1   +63.046, E3 -213493.011}
SPL {X  -150.233, Y  +726.516, Z    +0.000, E1   +62.565, E3 -213505.604}
SPL {X  -147.385, Y  +733.745, Z    +0.000, E1   +62.104, E3 -213515.908}
SPL {X  -144.667, Y  +739.825, Z    +0.000, E1   +61.658, E3 -213524.811}
SPL {X  -142.263, Y  +744.698, Z    +0.000, E1   +61.245, E3 -213532.126}
SPL {X  -138.935, Y  +750.833, Z    +0.000, E1   +60.711, E3 -213541.450}
SPL {X  -135.668, Y  +756.300, Z    +0.000, E1   +60.086, E3 -213550.014}
SPL {X  -132.995, Y  +760.433, Z    +0.000, E1   +59.601, E3 -213556.521}
SPL {X  -109.949, Y  +787.724, Z    +0.000, E1   +51.944, E3 -213649.083}
ENDSPLINE

SPLINE
SPL {X  -129.366, Y  +765.635, Z    +0.000, E1   +44.361, E3 -213758.825}
SPL {X  -144.719, Y  +739.715, Z    +0.000, E1   +37.620, E3 -213785.672}
SPL {X  -154.606, Y  +712.654, Z    +0.000, E1   +26.872, E3 -213798.892}
SPL {X  -158.229, Y  +695.175, Z    +0.000, E1   +17.621, E3 -213803.378}
SPL {X  -159.536, Y  +683.548, Z    +0.000, E1   +10.326, E3 -213805.166}
SPL {X  -159.946, Y  +675.243, Z    +0.000, E1    +4.608, E3 -213805.874}
SPL {X  -159.990, Y  +670.644, Z    +0.000, E1    +1.007, E3 -213806.050}
SPL {X  -159.990, Y  +669.188, Z    +0.000, E1    -0.261, E3 -213806.065}
SPL {X  -159.990, Y  +666.135, Z    +0.000, E1    -4.178, E3 -213806.154}
SPL {X  -159.990, Y  +662.249, Z    +0.000, E1   -10.338, E3 -213806.385}
SPL {X  -159.990, Y  +658.381, Z    +0.000, E1   -16.786, E3 -213806.777}
SPL {X  -159.990, Y  +651.878, Z    +0.000, E1   -27.298, E3 -213807.776}
SPL {X  -159.990, Y  +644.587, Z    +0.000, E1   -37.284, E3 -213809.358}
SPL {X  -159.990, Y  +633.621, Z    +0.000, E1   -47.309, E3 -213812.849}
SPL {X  -159.990, Y  +588.658, Z    +0.000, E1   -60.812, E3 -213835.169}
SPL {X  -159.990, Y  +495.038, Z    +0.000, E1   -63.580, E3 -213910.406}
SPL {X  -159.990, Y  +483.848, Z    +0.000, E1   -63.590, E3 -213922.190}
SPL {X  -159.990, Y  +471.874, Z    +0.000, E1   -63.586, E3 -213934.816}
SPL {X  -159.990, Y  +461.079, Z    +0.000, E1   -63.579, E3 -213946.225}
SPL {X  -159.990, Y  +450.188, Z    +0.000, E1   -63.581, E3 -213957.715}
SPL {X  -159.990, Y  +442.553, Z    +0.000, E1   -63.337, E3 -213967.539}
ENDSPLINE

SPLINE
SPL {X  -159.990, Y  +465.419, Z    +0.000, E1   -58.181, E3 -213976.384}
ENDSPLINE

SPLINE
SPL {X  -159.990, Y  +455.003, Z    +0.000, E1   -58.788, E3 -213985.922}
SPL {X  -159.990, Y  +443.180, Z    +0.000, E1   -59.522, E3 -213995.961}
SPL {X  -159.990, Y  +431.227, Z    +0.000, E1   -60.120, E3 -214006.653}
SPL {X  -159.990, Y  +418.989, Z    +0.000, E1   -60.714, E3 -214017.288}
SPL {X  -159.990, Y  +401.382, Z    +0.000, E1   -61.735, E3 -214030.757}
SPL {X  -159.983, Y  +381.042, Z    +0.000, E1   -62.802, E3 -214045.717}
SPL {X  -159.542, Y  +370.537, Z    +0.000, E1   -63.069, E3 -214055.099}
SPL {X  -158.758, Y  +362.683, Z    +0.000, E1   -62.956, E3 -214064.373}
SPL {X  -157.125, Y  +352.357, Z    +0.000, E1   -62.751, E3 -214077.106}
SPL {X  -154.421, Y  +340.656, Z    +0.000, E1   -62.344, E3 -214092.459}
SPL {X  -151.938, Y  +332.383, Z    +0.000, E1   -61.927, E3 -214103.932}
SPL {X  -149.604, Y  +325.796, Z    +0.000, E1   -61.568, E3 -214113.318}
SPL {X  -147.413, Y  +320.320, Z    +0.000, E1   -61.198, E3 -214121.371}
SPL {X  -145.235, Y  +315.391, Z    +0.000, E1   -60.847, E3 -214128.746}
SPL {X  -141.610, Y  +308.046, Z    +0.000, E1   -60.266, E3 -214139.982}
SPL {X  -138.010, Y  +301.568, Z    +0.000, E1   -59.585, E3 -214150.253}
SPL {X  -134.495, Y  +295.853, Z    +0.000, E1   -58.965, E3 -214159.391}
SPL {X  -113.541, Y  +269.782, Z    +0.000, E1   -50.113, E3 -214266.983}
ENDSPLINE

SPLINE
SPL {X  -145.506, Y  +315.982, Z    +0.000, E1   -36.457, E3 -214380.218}
SPL {X  -155.358, Y  +344.279, Z    +0.000, E1   -24.937, E3 -214394.643}
SPL {X  -158.582, Y  +361.322, Z    +0.000, E1   -15.773, E3 -214398.987}
SPL {X  -159.657, Y  +372.183, Z    +0.000, E1    -8.995, E3 -214400.595}
SPL {X  -159.986, Y  +381.348, Z    +0.000, E1    -2.678, E3 -214401.283}
SPL {X  -159.990, Y  +384.517, Z    +0.000, E1    -0.022, E3 -214401.373}
SPL {X  -159.990, Y  +385.713, Z    +0.000, E1    +1.275, E3 -214401.393}
SPL {X  -159.990, Y  +388.743, Z    +0.000, E1    +5.147, E3 -214401.523}
SPL {X  -159.990, Y  +393.154, Z    +0.000, E1   +11.942, E3 -214401.854}
SPL {X  -159.990, Y  +397.198, Z    +0.000, E1   +18.490, E3 -214402.352}
SPL {X  -159.990, Y  +402.771, Z    +0.000, E1   +27.045, E3 -214403.315}
SPL {X  -159.990, Y  +416.096, Z    +0.000, E1   +42.325, E3 -214406.982}
SPL {X  -159.990, Y  +469.763, Z    +0.000, E1   +60.937, E3 -214432.212}
SPL {X  -159.990, Y  +561.242, Z    +0.000, E1   +63.988, E3 -214503.160}
SPL {X  -159.990, Y  +574.019, Z    +0.000, E1   +64.020, E3 -214516.326}
SPL {X  -159.990, Y  +591.720, Z    +0.000, E1   +64.032, E3 -214534.625}
SPL {X  -159.990, Y  +605.088, Z    +0.000, E1   +63.988, E3 -214548.552}
SPL {X  -159.990, Y  +614.683, Z    +0.000, E1   +63.997, E3 -214558.447}
SPL {X  -159.990, Y  +629.274, Z    +0.000, E1   +64.033, E3 -214573.478}
SPL {X  -159.990, Y  +645.396, Z    +0.000, E1   +64.010, E3 -214590.209}
SPL {X  -159.990, Y  +656.294, Z    +0.000, E1   +63.988, E3 -214601.539}
SPL {X  -159.990, Y  +667.666, Z    +0.000, E1   +64.016, E3 -214613.230}
SPL {X  -159.767, Y  +679.937, Z    +0.000, E1   +63.968, E3 -214626.206}
SPL {X  -158.736, Y  +691.491, Z    +0.000, E1   +63.843, E3 -214639.204}
SPL {X  -157.131, Y  +701.612, Z    +0.000, E1   +63.591, E3 -214651.394}
SPL {X  -155.594, Y  +708.746, Z    +0.000, E1   +63.361, E3 -214660.374}
SPL {X  -153.286, Y  +717.329, Z    +0.000, E1   +63.046, E3 -214671.582}
SPL {X  -150.953, Y  +724.510, Z    +0.000, E1   +62.654, E3 -214681.410}
SPL {X  -148.087, Y  +732.056, Z    +0.000, E1   +62.252, E3 -214691.993}
SPL {X  -144.667, Y  +739.825, Z    +0.000, E1   +61.658, E3 -214703.382}
SPL {X  -142.263, Y  +744.698, Z    +0.000, E1   +61.245, E3 -214710.697}
SPL {X  -139.956, Y  +749.019, Z    +0.000, E1   +60.852, E3 -214717.275}
SPL {X  -136.617, Y  +754.762, Z    +0.000, E1   +60.296, E3 -214726.129}
SPL {X  -132.995, Y  +760.433, Z    +0.000, E1   +59.601, E3 -214735.093}
SPL {X  -109.949, Y  +787.724, Z    +0.000, E1   +51.944, E3 -214827.654}
ENDSPLINE

SPLINE
SPL {X  -129.366, Y  +765.635, Z    +0.000, E1   +44.361, E3 -214937.396}
SPL {X  -144.719, Y  +739.715, Z    +0.000, E1   +37.620, E3 -214964.244}
SPL {X  -154.606, Y  +712.654, Z    +0.000, E1   +26.872, E3 -214977.464}
SPL {X  -158.229, Y  +695.175, Z    +0.000, E1   +17.621, E3 -214981.950}
SPL {X  -159.735, Y  +680.532, Z    +0.000, E1    +8.352, E3 -214984.042}
SPL {X  -159.976, Y  +673.579, Z    +0.000, E1    +3.308, E3 -214984.536}
SPL {X  -159.990, Y  +669.438, Z    +0.000, E1    +0.061, E3 -214984.634}
SPL {X  -159.990, Y  +667.221, Z    +0.000, E1    -2.789, E3 -214984.677}
SPL {X  -159.990, Y  +663.611, Z    +0.000, E1    -7.967, E3 -214984.867}
SPL {X  -159.990, Y  +658.381, Z    +0.000, E1   -16.786, E3 -214985.348}
SPL {X  -159.990, Y  +651.878, Z    +0.000, E1   -27.298, E3 -214986.347}
SPL {X  -159.990, Y  +644.587, Z    +0.000, E1   -37.284, E3 -214987.930}
SPL {X  -159.990, Y  +633.621, Z    +0.000, E1   -47.309, E3 -214991.421}
SPL {X  -159.990, Y  +588.658, Z    +0.000, E1   -60.812, E3 -215013.741}
SPL {X  -159.990, Y  +495.038, Z    +0.000, E1   -63.580, E3 -215088.977}
SPL {X  -159.990, Y  +483.848, Z    +0.000, E1   -63.590, E3 -215100.762}
SPL {X  -159.990, Y  +471.874, Z    +0.000, E1   -63.586, E3 -215113.387}
SPL {X  -159.990, Y  +461.079, Z    +0.000, E1   -63.579, E3 -215124.796}
SPL {X  -159.990, Y  +450.188, Z    +0.000, E1   -63.581, E3 -215136.287}
SPL {X  -159.990, Y  +442.553, Z    +0.000, E1   -63.337, E3 -215146.110}
ENDSPLINE

SPLINE
SPL {X  -159.990, Y  +465.419, Z    +0.000, E1   -58.181, E3 -215154.956}
ENDSPLINE

SPLINE
SPL {X  -159.990, Y  +455.003, Z    +0.000, E1   -58.788, E3 -215164.494}
SPL {X  -159.990, Y  +443.180, Z    +0.000, E1   -59.522, E3 -215174.532}
SPL {X  -159.990, Y  +431.227, Z    +0.000, E1   -60.120, E3 -215185.224}
SPL {X  -159.990, Y  +418.989, Z    +0.000, E1   -60.714, E3 -215195.859}
SPL {X  -159.990, Y  +401.382, Z    +0.000, E1   -61.735, E3 -215209.329}
SPL {X  -159.983, Y  +381.042, Z    +0.000, E1   -62.802, E3 -215224.288}
SPL {X  -159.542, Y  +370.537, Z    +0.000, E1   -63.069, E3 -215233.670}
SPL {X  -158.287, Y  +359.218, Z    +0.000, E1   -62.927, E3 -215247.085}
SPL {X  -155.813, Y  +346.180, Z    +0.000, E1   -62.560, E3 -215263.662}
SPL {X  -152.656, Y  +334.615, Z    +0.000, E1   -62.078, E3 -215279.314}
SPL {X  -149.604, Y  +325.796, Z    +0.000, E1   -61.568, E3 -215291.889}
SPL {X  -147.413, Y  +320.320, Z    +0.000, E1   -61.198, E3 -215299.942}
SPL {X  -145.235, Y  +315.391, Z    +0.000, E1   -60.847, E3 -215307.317}
SPL {X  -142.998, Y  +310.747, Z    +0.000, E1   -60.455, E3 -215314.430}
SPL {X  -140.747, Y  +306.427, Z    +0.000, E1   -60.074, E3 -215321.139}
SPL {X  -138.010, Y  +301.568, Z    +0.000, E1   -59.585, E3 -215328.825}
SPL {X  -134.495, Y  +295.853, Z    +0.000, E1   -58.965, E3 -215337.962}
SPL {X  -113.541, Y  +269.782, Z    +0.000, E1   -50.113, E3 -215445.554}
ENDSPLINE

SPLINE
SPL {X  -141.985, Y  +308.763, Z    +0.000, E1   -38.695, E3 -215553.507}
SPL {X  -154.491, Y  +340.913, Z    +0.000, E1   -26.570, E3 -215571.959}
SPL {X  -158.582, Y  +361.322, Z    +0.000, E1   -15.773, E3 -215577.558}
SPL {X  -159.657, Y  +372.183, Z    +0.000, E1    -8.995, E3 -215579.166}
SPL {X  -159.949, Y  +378.873, Z    +0.000, E1    -4.398, E3 -215579.740}
SPL {X  -159.990, Y  +384.063, Z    +0.000, E1    -0.515, E3 -215579.936}
SPL {X  -159.990, Y  +386.497, Z    +0.000, E1    +2.123, E3 -215579.992}
SPL {X  -159.990, Y  +389.673, Z    +0.000, E1    +6.604, E3 -215580.145}
SPL {X  -159.990, Y  +394.848, Z    +0.000, E1   +14.441, E3 -215580.634}
SPL {X  -159.990, Y  +402.771, Z    +0.000, E1   +27.045, E3 -215581.886}
SPL {X  -159.990, Y  +414.719, Z    +0.000, E1   +41.161, E3 -215585.060}
SPL {X  -159.990, Y  +424.336, Z    +0.000, E1   +48.481, E3 -215588.495}
SPL {X  -159.990, Y  +469.763, Z    +0.000, E1   +60.937, E3 -215610.783}
SPL {X  -159.990, Y  +561.242, Z    +0.000, E1   +63.988, E3 -215681.732}
SPL {X  -159.990, Y  +574.019, Z    +0.000, E1   +64.020, E3 -215694.898}
SPL {X  -159.990, Y  +588.139, Z    +0.000, E1   +64.000, E3 -215709.546}
SPL {X  -159.990, Y  +601.786, Z    +0.000, E1   +64.016, E3 -215723.650}
SPL {X  -159.990, Y  +614.683, Z    +0.000, E1   +63.997, E3 -215737.018}
SPL {X  -159.990, Y  +629.274, Z    +0.000, E1   +64.033, E3 -215752.049}
SPL {X  -159.990, Y  +645.396, Z    +0.000, E1   +64.010, E3 -215768.780}
SPL {X  -159.990, Y  +656.294, Z    +0.000, E1   +63.988, E3 -215780.110}
SPL {X  -159.990, Y  +667.666, Z    +0.000, E1   +64.016, E3 -215791.802}
SPL {X  -159.767, Y  +679.937, Z    +0.000, E1   +63.968, E3 -215804.777}
SPL {X  -158.736, Y  +691.491, Z    +0.000, E1   +63.843, E3 -215817.775}
SPL {X  -157.131, Y  +701.612, Z    +0.000, E1   +63.591, E3 -215829.965}
SPL {X  -154.918, Y  +711.464, Z    +0.000, E1   +63.294, E3 -215842.401}
SPL {X  -152.656, Y  +719.385, Z    +0.000, E1   +62.921, E3 -215852.969}
SPL {X  -150.233, Y  +726.516, Z    +0.000, E1   +62.565, E3 -215862.747}
SPL {X  -147.385, Y  +733.745, Z    +0.000, E1   +62.104, E3 -215873.051}
SPL {X  -144.667, Y  +739.825, Z    +0.000, E1   +61.658, E3 -215881.953}
SPL {X  -142.263, Y  +744.698, Z    +0.000, E1   +61.245, E3 -215889.269}
SPL {X  -138.935, Y  +750.833, Z    +0.000, E1   +60.711, E3 -215898.593}
SPL {X  -135.668, Y  +756.300, Z    +0.000, E1   +60.086, E3 -215907.156}
SPL {X  -132.995, Y  +760.433, Z    +0.000, E1   +59.601, E3 -215913.664}
SPL {X  -109.949, Y  +787.724, Z    +0.000, E1   +51.944, E3 -216006.226}
ENDSPLINE

SPLINE
SPL {X  -129.366, Y  +765.635, Z    +0.000, E1   +44.361, E3 -216115.968}
SPL {X  -144.719, Y  +739.715, Z    +0.000, E1   +37.620, E3 -216142.815}
SPL {X  -154.606, Y  +712.654, Z    +0.000, E1   +26.872, E3 -216156.035}
SPL {X  -158.229, Y  +695.175, Z    +0.000, E1   +17.621, E3 -216160.521}
SPL {X  -159.735, Y  +680.532, Z    +0.000, E1    +8.352, E3 -216162.613}
SPL {X  -159.976, Y  +673.579, Z    +0.000, E1    +3.308, E3 -216163.108}
SPL {X  -159.990, Y  +669.438, Z    +0.000, E1    +0.061, E3 -216163.205}
SPL {X  -159.990, Y  +666.135, Z    +0.000, E1    -4.178, E3 -216163.296}
SPL {X  -159.990, Y  +662.249, Z    +0.000, E1   -10.338, E3 -216163.528}
SPL {X  -159.990, Y  +658.381, Z    +0.000, E1   -16.786, E3 -216163.919}
SPL {X  -159.990, Y  +651.878, Z    +0.000, E1   -27.298, E3 -216164.918}
SPL {X  -159.990, Y  +644.587, Z    +0.000, E1   -37.284, E3 -216166.501}
SPL {X  -159.990, Y  +633.621, Z    +0.000, E1   -47.309, E3 -216169.992}
SPL {X  -159.990, Y  +588.658, Z    +0.000, E1   -60.812, E3 -216192.312}
SPL {X  -159.990, Y  +495.038, Z    +0.000, E1   -63.580, E3 -216267.548}
SPL {X  -159.990, Y  +483.848, Z    +0.000, E1   -63.590, E3 -216279.333}
SPL {X  -159.990, Y  +471.874, Z    +0.000, E1   -63.586, E3 -216291.959}
SPL {X  -159.990, Y  +461.079, Z    +0.000, E1   -63.579, E3 -216303.367}
SPL {X  -159.990, Y  +450.188, Z    +0.000, E1   -63.581, E3 -216314.858}
SPL {X  -159.990, Y  +442.553, Z    +0.000, E1   -63.337, E3 -216324.682}
ENDSPLINE

SPLINE
SPL {X  -159.990, Y  +465.419, Z    +0.000, E1   -58.181, E3 -216333.527}
ENDSPLINE

SPLINE
SPL {X  -159.990, Y  +455.003, Z    +0.000, E1   -58.788, E3 -216343.065}
SPL {X  -159.990, Y  +443.180, Z    +0.000, E1   -59.522, E3 -216353.103}
SPL {X  -159.990, Y  +431.227, Z    +0.000, E1   -60.120, E3 -216363.796}
SPL {X  -159.990, Y  +413.464, Z    +0.000, E1   -61.043, E3 -216378.786}
SPL {X  -159.990, Y  +395.417, Z    +0.000, E1   -62.063, E3 -216392.228}
SPL {X  -159.983, Y  +381.042, Z    +0.000, E1   -62.802, E3 -216402.860}
SPL {X  -159.542, Y  +370.537, Z    +0.000, E1   -63.069, E3 -216412.242}
SPL {X  -158.287, Y  +359.218, Z    +0.000, E1   -62.927, E3 -216425.657}
SPL {X  -156.553, Y  +349.515, Z    +0.000, E1   -62.627, E3 -216437.968}
SPL {X  -154.421, Y  +340.656, Z    +0.000, E1   -62.344, E3 -216449.602}
SPL {X  -151.938, Y  +332.383, Z    +0.000, E1   -61.927, E3 -216461.075}
SPL {X  -149.604, Y  +325.796, Z    +0.000, E1   -61.568, E3 -216470.461}
SPL {X  -147.413, Y  +320.320, Z    +0.000, E1   -61.198, E3 -216478.514}
SPL {X  -145.235, Y  +315.391, Z    +0.000, E1   -60.847, E3 -216485.888}
SPL {X  -141.610, Y  +308.046, Z    +0.000, E1   -60.266, E3 -216497.125}
SPL {X  -138.010, Y  +301.568, Z    +0.000, E1   -59.585, E3 -216507.396}
SPL {X  -134.495, Y  +295.853, Z    +0.000, E1   -58.965, E3 -216516.533}
SPL {X  -113.541, Y  +269.782, Z    +0.000, E1   -50.113, E3 -216624.126}
ENDSPLINE

SPLINE
SPL {X  -141.985, Y  +308.763, Z    +0.000, E1   -38.695, E3 -216732.078}
SPL {X  -154.491, Y  +340.913, Z    +0.000, E1   -26.570, E3 -216750.531}
SPL {X  -158.582, Y  +361.322, Z    +0.000, E1   -15.773, E3 -216756.129}
SPL {X  -159.657, Y  +372.183, Z    +0.000, E1    -8.995, E3 -216757.738}
SPL {X  -159.949, Y  +378.873, Z    +0.000, E1    -4.398, E3 -216758.312}
SPL {X  -159.990, Y  +384.063, Z    +0.000, E1    -0.515, E3 -216758.508}
SPL {X  -159.990, Y  +386.497, Z    +0.000, E1    +2.123, E3 -216758.564}
SPL {X  -159.990, Y  +391.572, Z    +0.000, E1    +9.236, E3 -216758.870}
SPL {X  -159.990, Y  +397.198, Z    +0.000, E1   +18.490, E3 -216759.494}
SPL {X  -159.990, Y  +402.771, Z    +0.000, E1   +27.045, E3 -216760.458}
SPL {X  -159.990, Y  +416.096, Z    +0.000, E1   +42.325, E3 -216764.125}
SPL {X  -159.990, Y  +469.763, Z    +0.000, E1   +60.937, E3 -216789.355}
SPL {X  -159.990, Y  +565.969, Z    +0.000, E1   +64.023, E3 -216865.129}
SPL {X  -159.990, Y  +578.082, Z    +0.000, E1   +63.987, E3 -216877.737}
SPL {X  -159.990, Y  +588.139, Z    +0.000, E1   +64.000, E3 -216888.117}
SPL {X  -159.990, Y  +601.786, Z    +0.000, E1   +64.016, E3 -216902.221}
SPL {X  -159.990, Y  +618.770, Z    +0.000, E1   +64.031, E3 -216919.757}
SPL {X  -159.990, Y  +636.111, Z    +0.000, E1   +64.024, E3 -216937.712}
SPL {X  -159.990, Y  +652.385, Z    +0.000, E1   +64.020, E3 -216954.570}
SPL {X  -159.990, Y  +667.666, Z    +0.000, E1   +64.016, E3 -216970.373}
SPL {X  -159.767, Y  +679.937, Z    +0.000, E1   +63.968, E3 -216983.348}
SPL {X  -159.113, Y  +688.225, Z    +0.000, E1   +63.867, E3 -216992.626}
SPL {X  -158.361, Y  +694.273, Z    +0.000, E1   +63.762, E3 -216999.664}
SPL {X  -157.131, Y  +701.612, Z    +0.000, E1   +63.591, E3 -217008.537}
SPL {X  -154.918, Y  +711.464, Z    +0.000, E1   +63.294, E3 -217020.972}
SPL {X  -151.874, Y  +721.810, Z    +0.000, E1   +62.834, E3 -217034.779}
SPL {X  -148.087, Y  +732.056, Z    +0.000, E1   +62.252, E3 -217049.135}
SPL {X  -144.667, Y  +739.825, Z    +0.000, E1   +61.658, E3 -217060.525}
SPL {X  -142.263, Y  +744.698, Z    +0.000, E1   +61.245, E3 -217067.840}
SPL {X  -138.935, Y  +750.833, Z    +0.000, E1   +60.711, E3 -217077.165}
SPL {X  -135.668, Y  +756.300, Z    +0.000, E1   +60.086, E3 -217085.728}
SPL {X  -132.995, Y  +760.433, Z    +0.000, E1   +59.601, E3 -217092.235}
SPL {X  -109.949, Y  +787.724, Z    +0.000, E1   +51.944, E3 -217184.797}
ENDSPLINE

SPLINE
SPL {X  -129.366, Y  +765.635, Z    +0.000, E1   +44.361, E3 -217294.539}
SPL {X  -144.719, Y  +739.715, Z    +0.000, E1   +37.620, E3 -217321.386}
SPL {X  -154.606, Y  +712.654, Z    +0.000, E1   +26.872, E3 -217334.606}
SPL {X  -158.229, Y  +695.175, Z    +0.000, E1   +17.621, E3 -217339.092}
SPL {X  -159.735, Y  +680.532, Z    +0.000, E1    +8.352, E3 -217341.185}
SPL {X  -159.990, Y  +671.731, Z    +0.000, E1    +1.953, E3 -217341.735}
SPL {X  -159.990, Y  +668.624, Z    +0.000, E1    -0.752, E3 -217341.791}
SPL {X  -159.990, Y  +663.611, Z    +0.000, E1    -7.967, E3 -217342.010}
SPL {X  -159.990, Y  +658.381, Z    +0.000, E1   -16.786, E3 -217342.491}
SPL {X  -159.990, Y  +651.878, Z    +0.000, E1   -27.298, E3 -217343.490}
SPL {X  -159.990, Y  +644.587, Z    +0.000, E1   -37.284, E3 -217345.073}
SPL {X  -159.990, Y  +633.621, Z    +0.000, E1   -47.309, E3 -217348.564}
SPL {X  -159.990, Y  +588.658, Z    +0.000, E1   -60.812, E3 -217370.884}
SPL {X  -159.990, Y  +495.038, Z    +0.000, E1   -63.580, E3 -217446.120}
SPL {X  -159.990, Y  +483.848, Z    +0.000, E1   -63.590, E3 -217457.905}
SPL {X  -159.990, Y  +471.874, Z    +0.000, E1   -63.586, E3 -217470.530}
SPL {X  -159.990, Y  +461.079, Z    +0.000, E1   -63.579, E3 -217481.939}
SPL {X  -159.990, Y  +450.188, Z    +0.000, E1   -63.581, E3 -217493.429}
SPL {X  -159.990, Y  +442.553, Z    +0.000, E1   -63.337, E3 -217503.253}
ENDSPLINE

SPLINE
SPL {X  -159.990, Y  +465.419, Z    +0.000, E1   -58.181, E3 -217512.098}
ENDSPLINE

SPLINE
SPL {X  -159.990, Y  +455.003, Z    +0.000, E1   -58.788, E3 -217521.637}
SPL {X  -159.990, Y  +443.180, Z    +0.000, E1   -59.522, E3 -217531.675}
SPL {X  -159.990, Y  +431.227, Z    +0.000, E1   -60.120, E3 -217542.367}
SPL {X  -159.990, Y  +413.464, Z    +0.000, E1   -61.043, E3 -217557.357}
SPL {X  -159.990, Y  +395.417, Z    +0.000, E1   -62.063, E3 -217570.800}
SPL {X  -159.983, Y  +381.042, Z    +0.000, E1   -62.802, E3 -217581.431}
SPL {X  -159.542, Y  +370.537, Z    +0.000, E1   -63.069, E3 -217590.813}
SPL {X  -158.758, Y  +362.683, Z    +0.000, E1   -62.956, E3 -217600.087}
SPL {X  -157.125, Y  +352.357, Z    +0.000, E1   -62.751, E3 -217612.820}
SPL {X  -154.421, Y  +340.656, Z    +0.000, E1   -62.344, E3 -217628.173}
SPL {X  -151.938, Y  +332.383, Z    +0.000, E1   -61.927, E3 -217639.646}
SPL {X  -149.604, Y  +325.796, Z    +0.000, E1   -61.568, E3 -217649.032}
SPL {X  -147.413, Y  +320.320, Z    +0.000, E1   -61.198, E3 -217657.085}
SPL {X  -145.235, Y  +315.391, Z    +0.000, E1   -60.847, E3 -217664.460}
SPL {X  -141.610, Y  +308.046, Z    +0.000, E1   -60.266, E3 -217675.696}
SPL {X  -138.010, Y  +301.568, Z    +0.000, E1   -59.585, E3 -217685.967}
SPL {X  -134.495, Y  +295.853, Z    +0.000, E1   -58.965, E3 -217695.105}
SPL {X  -113.541, Y  +269.782, Z    +0.000, E1   -50.113, E3 -217802.697}
ENDSPLINE

SPLINE
SPL {X  -141.985, Y  +308.763, Z    +0.000, E1   -38.695, E3 -217910.650}
SPL {X  -154.491, Y  +340.913, Z    +0.000, E1   -26.570, E3 -217929.102}
SPL {X  -158.582, Y  +361.322, Z    +0.000, E1   -15.773, E3 -217934.701}
SPL {X  -159.657, Y  +372.183, Z    +0.000, E1    -8.995, E3 -217936.309}
SPL {X  -159.949, Y  +378.873, Z    +0.000, E1    -4.398, E3 -217936.883}
SPL {X  -159.990, Y  +384.063, Z    +0.000, E1    -0.515, E3 -217937.079}
SPL {X  -159.990, Y  +386.497, Z    +0.000, E1    +2.123, E3 -217937.135}
SPL {X  -159.990, Y  +389.673, Z    +0.000, E1    +6.604, E3 -217937.288}
SPL {X  -159.990, Y  +394.848, Z    +0.000, E1   +14.441, E3 -217937.777}
SPL {X  -159.990, Y  +402.771, Z    +0.000, E1   +27.045, E3 -217939.029}
SPL {X  -159.990, Y  +414.719, Z    +0.000, E1   +41.161, E3 -217942.203}
SPL {X  -159.990, Y  +424.336, Z    +0.000, E1   +48.481, E3 -217945.638}
SPL {X  -159.990, Y  +469.763, Z    +0.000, E1   +60.937, E3 -217967.926}
SPL {X  -159.990, Y  +561.242, Z    +0.000, E1   +63.988, E3 -218038.875}
SPL {X  -159.990, Y  +574.019, Z    +0.000, E1   +64.020, E3 -218052.041}
SPL {X  -159.990, Y  +588.139, Z    +0.000, E1   +64.000, E3 -218066.689}
SPL {X  -159.990, Y  +601.786, Z    +0.000, E1   +64.016, E3 -218080.793}
SPL {X  -159.990, Y  +614.683, Z    +0.000, E1   +63.997, E3 -218094.161}
SPL {X  -159.990, Y  +629.274, Z    +0.000, E1   +64.033, E3 -218109.192}
SPL {X  -159.990, Y  +645.396, Z    +0.000, E1   +64.010, E3 -218125.923}
SPL {X  -159.990, Y  +656.294, Z    +0.000, E1   +63.988, E3 -218137.253}
SPL {X  -159.990, Y  +667.666, Z    +0.000, E1   +64.016, E3 -218148.945}
SPL {X  -159.767, Y  +679.937, Z    +0.000, E1   +63.968, E3 -218161.920}
SPL {X  -158.736, Y  +691.491, Z    +0.000, E1   +63.843, E3 -218174.918}
SPL {X  -157.131, Y  +701.612, Z    +0.000, E1   +63.591, E3 -218187.108}
SPL {X  -154.918, Y  +711.464, Z    +0.000, E1   +63.294, E3 -218199.543}
SPL {X  -152.656, Y  +719.385, Z    +0.000, E1   +62.921, E3 -218210.112}
SPL {X  -150.233, Y  +726.516, Z    +0.000, E1   +62.565, E3 -218219.890}
SPL {X  -147.385, Y  +733.745, Z    +0.000, E1   +62.104, E3 -218230.194}
SPL {X  -144.667, Y  +739.825, Z    +0.000, E1   +61.658, E3 -218239.096}
SPL {X  -142.263, Y  +744.698, Z    +0.000, E1   +61.245, E3 -218246.412}
SPL {X  -138.935, Y  +750.833, Z    +0.000, E1   +60.711, E3 -218255.736}
SPL {X  -135.668, Y  +756.300, Z    +0.000, E1   +60.086, E3 -218264.299}
SPL {X  -132.995, Y  +760.433, Z    +0.000, E1   +59.601, E3 -218270.807}
SPL {X  -109.949, Y  +787.724, Z    +0.000, E1   +51.944, E3 -218363.368}
ENDSPLINE

SPLINE
SPL {X  -129.366, Y  +765.635, Z    +0.000, E1   +44.361, E3 -218473.110}
SPL {X  -144.719, Y  +739.715, Z    +0.000, E1   +37.620, E3 -218499.958}
SPL {X  -154.606, Y  +712.654, Z    +0.000, E1   +26.872, E3 -218513.178}
SPL {X  -158.229, Y  +695.175, Z    +0.000, E1   +17.621, E3 -218517.664}
SPL {X  -159.735, Y  +680.532, Z    +0.000, E1    +8.352, E3 -218519.756}
SPL {X  -159.976, Y  +673.579, Z    +0.000, E1    +3.308, E3 -218520.250}
SPL {X  -159.990, Y  +669.438, Z    +0.000, E1    +0.061, E3 -218520.348}
SPL {X  -159.990, Y  +666.135, Z    +0.000, E1    -4.178, E3 -218520.439}
SPL {X  -159.990, Y  +662.249, Z    +0.000, E1   -10.338, E3 -218520.671}
SPL {X  -159.990, Y  +658.381, Z    +0.000, E1   -16.786, E3 -218521.062}
SPL {X  -159.990, Y  +651.878, Z    +0.000, E1   -27.298, E3 -218522.061}
SPL {X  -159.990, Y  +644.587, Z    +0.000, E1   -37.284, E3 -218523.644}
SPL {X  -159.990, Y  +633.621, Z    +0.000, E1   -47.309, E3 -218527.135}
SPL {X  -159.990, Y  +588.658, Z    +0.000, E1   -60.812, E3 -218549.455}
SPL {X  -159.990, Y  +495.038, Z    +0.000, E1   -63.580, E3 -218624.691}
SPL {X  -159.990, Y  +483.848, Z    +0.000, E1   -63.590, E3 -218636.476}
SPL {X  -159.990, Y  +471.874, Z    +0.000, E1   -63.586, E3 -218649.102}
SPL {X  -159.990, Y  +461.079, Z    +0.000, E1   -63.579, E3 -218660.510}
SPL {X  -159.990, Y  +450.188, Z    +0.000, E1   -63.581, E3 -218672.001}
SPL {X  -159.990, Y  +442.553, Z    +0.000, E1   -63.337, E3 -218681.824}
ENDSPLINE

SPLINE
SPL {X  -159.990, Y  +465.419, Z    +0.000, E1   -58.181, E3 -218690.670}
ENDSPLINE

SPLINE
SPL {X  -159.990, Y  +455.003, Z    +0.000, E1   -58.788, E3 -218700.208}
SPL {X  -159.990, Y  +443.180, Z    +0.000, E1   -59.522, E3 -218710.246}
SPL {X  -159.990, Y  +431.227, Z    +0.000, E1   -60.120, E3 -218720.938}
SPL {X  -159.990, Y  +413.464, Z    +0.000, E1   -61.043, E3 -218735.928}
SPL {X  -159.990, Y  +395.417, Z    +0.000, E1   -62.063, E3 -218749.371}
SPL {X  -159.983, Y  +381.042, Z    +0.000, E1   -62.802, E3 -218760.003}
SPL {X  -159.542, Y  +370.537, Z    +0.000, E1   -63.069, E3 -218769.385}
SPL {X  -158.287, Y  +359.218, Z    +0.000, E1   -62.927, E3 -218782.799}
SPL {X  -156.553, Y  +349.515, Z    +0.000, E1   -62.627, E3 -218795.111}
SPL {X  -154.421, Y  +340.656, Z    +0.000, E1   -62.344, E3 -218806.745}
SPL {X  -151.938, Y  +332.383, Z    +0.000, E1   -61.927, E3 -218818.218}
SPL {X  -149.604, Y  +325.796, Z    +0.000, E1   -61.568, E3 -218827.603}
SPL {X  -147.413, Y  +320.320, Z    +0.000, E1   -61.198, E3 -218835.657}
SPL {X  -145.235, Y  +315.391, Z    +0.000, E1   -60.847, E3 -218843.031}
SPL {X  -141.610, Y  +308.046, Z    +0.000, E1   -60.266, E3 -218854.268}
SPL {X  -138.010, Y  +301.568, Z    +0.000, E1   -59.585, E3 -218864.539}
SPL {X  -134.495, Y  +295.853, Z    +0.000, E1   -58.965, E3 -218873.676}
SPL {X  -113.541, Y  +269.782, Z    +0.000, E1   -50.113, E3 -218981.269}
ENDSPLINE

SPLINE
SPL {X  -141.985, Y  +308.763, Z    +0.000, E1   -38.695, E3 -219089.221}
SPL {X  -154.491, Y  +340.913, Z    +0.000, E1   -26.570, E3 -219107.674}
SPL {X  -158.582, Y  +361.322, Z    +0.000, E1   -15.773, E3 -219113.272}
SPL {X  -159.657, Y  +372.183, Z    +0.000, E1    -8.995, E3 -219114.880}
SPL {X  -159.949, Y  +378.873, Z    +0.000, E1    -4.398, E3 -219115.455}
SPL {X  -159.990, Y  +384.063, Z    +0.000, E1    -0.515, E3 -219115.651}
SPL {X  -159.990, Y  +386.497, Z    +0.000, E1    +2.123, E3 -219115.707}
SPL {X  -159.990, Y  +391.572, Z    +0.000, E1    +9.236, E3 -219116.013}
SPL {X  -159.990, Y  +397.198, Z    +0.000, E1   +18.490, E3 -219116.637}
SPL {X  -159.990, Y  +402.771, Z    +0.000, E1   +27.045, E3 -219117.601}
SPL {X  -159.990, Y  +416.096, Z    +0.000, E1   +42.325, E3 -219121.268}
SPL {X  -159.990, Y  +469.763, Z    +0.000, E1   +60.937, E3 -219146.498}
SPL {X  -159.990, Y  +565.969, Z    +0.000, E1   +64.023, E3 -219222.272}
SPL {X  -159.990, Y  +578.082, Z    +0.000, E1   +63.987, E3 -219234.880}
SPL {X  -159.990, Y  +588.139, Z    +0.000, E1   +64.000, E3 -219245.260}
SPL {X  -159.990, Y  +601.786, Z    +0.000, E1   +64.016, E3 -219259.364}
SPL {X  -159.990, Y  +618.770, Z    +0.000, E1   +64.031, E3 -219276.900}
SPL {X  -159.990, Y  +636.111, Z    +0.000, E1   +64.024, E3 -219294.855}
SPL {X  -159.990, Y  +652.385, Z    +0.000, E1   +64.020, E3 -219311.713}
SPL {X  -159.990, Y  +667.666, Z    +0.000, E1   +64.016, E3 -219327.516}
SPL {X  -159.767, Y  +679.937, Z    +0.000, E1   +63.968, E3 -219340.491}
SPL {X  -159.113, Y  +688.225, Z    +0.000, E1   +63.867, E3 -219349.769}
SPL {X  -158.361, Y  +694.273, Z    +0.000, E1   +63.762, E3 -219356.807}
SPL {X  -157.131, Y  +701.612, Z    +0.000, E1   +63.591, E3 -219365.680}
SPL {X  -155.594, Y  +708.746, Z    +0.000, E1   +63.361, E3 -219374.660}
SPL {X  -153.286, Y  +717.329, Z    +0.000, E1   +63.046, E3 -219385.868}
SPL {X  -150.233, Y  +726.516, Z    +0.000, E1   +62.565, E3 -219398.461}
SPL {X  -147.385, Y  +733.745, Z    +0.000, E1   +62.104, E3 -219408.766}
SPL {X  -144.667, Y  +739.825, Z    +0.000, E1   +61.658, E3 -219417.668}
SPL {X  -142.263, Y  +744.698, Z    +0.000, E1   +61.245, E3 -219424.983}
SPL {X  -138.935, Y  +750.833, Z    +0.000, E1   +60.711, E3 -219434.307}
SPL {X  -135.668, Y  +756.300, Z    +0.000, E1   +60.086, E3 -219442.871}
SPL {X  -132.995, Y  +760.433, Z    +0.000, E1   +59.601, E3 -219449.378}
SPL {X  -109.949, Y  +787.724, Z    +0.000, E1   +51.944, E3 -219541.940}
ENDSPLINE

SPLINE
SPL {X  -129.366, Y  +765.635, Z    +0.000, E1   +44.361, E3 -219651.682}
SPL {X  -144.719, Y  +739.715, Z    +0.000, E1   +37.620, E3 -219678.529}
SPL {X  -154.606, Y  +712.654, Z    +0.000, E1   +26.872, E3 -219691.749}
SPL {X  -158.229, Y  +695.175, Z    +0.000, E1   +17.621, E3 -219696.235}
SPL {X  -159.536, Y  +683.548, Z    +0.000, E1   +10.326, E3 -219698.023}
SPL {X  -159.946, Y  +675.243, Z    +0.000, E1    +4.608, E3 -219698.732}
SPL {X  -159.990, Y  +670.644, Z    +0.000, E1    +1.007, E3 -219698.907}
SPL {X  -159.990, Y  +669.188, Z    +0.000, E1    -0.261, E3 -219698.922}
SPL {X  -159.990, Y  +666.135, Z    +0.000, E1    -4.178, E3 -219699.011}
SPL {X  -159.990, Y  +662.249, Z    +0.000, E1   -10.338, E3 -219699.242}
SPL {X  -159.990, Y  +658.381, Z    +0.000, E1   -16.786, E3 -219699.634}
SPL {X  -159.990, Y  +651.878, Z    +0.000, E1   -27.298, E3 -219700.633}
SPL {X  -159.990, Y  +644.587, Z    +0.000, E1   -37.284, E3 -219702.216}
SPL {X  -159.990, Y  +633.621, Z    +0.000, E1   -47.309, E3 -219705.707}
SPL {X  -159.990, Y  +588.658, Z    +0.000, E1   -60.812, E3 -219728.026}
SPL {X  -159.990, Y  +495.038, Z    +0.000, E1   -63.580, E3 -219803.263}
SPL {X  -159.990, Y  +483.848, Z    +0.000, E1   -63.590, E3 -219815.047}
SPL {X  -159.990, Y  +471.874, Z    +0.000, E1   -63.586, E3 -219827.673}
SPL {X  -159.990, Y  +461.079, Z    +0.000, E1   -63.579, E3 -219839.082}
SPL {X  -159.990, Y  +450.188, Z    +0.000, E1   -63.581, E3 -219850.572}
SPL {X  -159.990, Y  +442.553, Z    +0.000, E1   -63.337, E3 -219860.396}
ENDSPLINE

SPLINE
SPL {X  -159.990, Y  +465.419, Z    +0.000, E1   -58.181, E3 -219869.241}
ENDSPLINE

SPLINE
SPL {X  -159.990, Y  +455.003, Z    +0.000, E1   -58.788, E3 -219878.779}
SPL {X  -159.990, Y  +443.180, Z    +0.000, E1   -59.522, E3 -219888.818}
SPL {X  -159.990, Y  +431.227, Z    +0.000, E1   -60.120, E3 -219899.510}
SPL {X  -159.990, Y  +418.989, Z    +0.000, E1   -60.714, E3 -219910.145}
SPL {X  -159.990, Y  +401.382, Z    +0.000, E1   -61.735, E3 -219923.614}
SPL {X  -159.983, Y  +381.042, Z    +0.000, E1   -62.802, E3 -219938.574}
SPL {X  -159.542, Y  +370.537, Z    +0.000, E1   -63.069, E3 -219947.956}
SPL {X  -158.758, Y  +362.683, Z    +0.000, E1   -62.956, E3 -219957.230}
SPL {X  -157.125, Y  +352.357, Z    +0.000, E1   -62.751, E3 -219969.963}
SPL {X  -154.421, Y  +340.656, Z    +0.000, E1   -62.344, E3 -219985.316}
SPL {X  -151.938, Y  +332.383, Z    +0.000, E1   -61.927, E3 -219996.789}
SPL {X  -149.604, Y  +325.796, Z    +0.000, E1   -61.568, E3 -220006.175}
SPL {X  -147.413, Y  +320.320, Z    +0.000, E1   -61.198, E3 -220014.228}
SPL {X  -145.235, Y  +315.391, Z    +0.000, E1   -60.847, E3 -220021.603}
SPL {X  -141.610, Y  +308.046, Z    +0.000, E1   -60.266, E3 -220032.839}
SPL {X  -138.010, Y  +301.568, Z    +0.000, E1   -59.585, E3 -220043.110}
SPL {X  -134.495, Y  +295.853, Z    +0.000, E1   -58.965, E3 -220052.248}
SPL {X  -113.541, Y  +269.782, Z    +0.000, E1   -50.113, E3 -220159.840}
ENDSPLINE

SPLINE
SPL {X  -145.506, Y  +315.982, Z    +0.000, E1   -36.457, E3 -220273.076}
SPL {X  -155.358, Y  +344.279, Z    +0.000, E1   -24.937, E3 -220287.500}
SPL {X  -158.582, Y  +361.322, Z    +0.000, E1   -15.773, E3 -220291.844}
SPL {X  -159.657, Y  +372.183, Z    +0.000, E1    -8.995, E3 -220293.452}
SPL {X  -159.986, Y  +381.348, Z    +0.000, E1    -2.678, E3 -220294.140}
SPL {X  -159.990, Y  +384.517, Z    +0.000, E1    -0.022, E3 -220294.230}
SPL {X  -159.990, Y  +385.713, Z    +0.000, E1    +1.275, E3 -220294.250}
SPL {X  -159.990, Y  +388.743, Z    +0.000, E1    +5.147, E3 -220294.380}
SPL {X  -159.990, Y  +393.154, Z    +0.000, E1   +11.942, E3 -220294.712}
SPL {X  -159.990, Y  +397.198, Z    +0.000, E1   +18.490, E3 -220295.209}
SPL {X  -159.990, Y  +402.771, Z    +0.000, E1   +27.045, E3 -220296.172}
SPL {X  -159.990, Y  +416.096, Z    +0.000, E1   +42.325, E3 -220299.839}
SPL {X  -159.990, Y  +469.763, Z    +0.000, E1   +60.937, E3 -220325.069}
SPL {X  -159.990, Y  +561.242, Z    +0.000, E1   +63.988, E3 -220396.017}
SPL {X  -159.990, Y  +574.019, Z    +0.000, E1   +64.020, E3 -220409.184}
SPL {X  -159.990, Y  +591.720, Z    +0.000, E1   +64.032, E3 -220427.482}
SPL {X  -159.990, Y  +605.088, Z    +0.000, E1   +63.988, E3 -220441.409}
SPL {X  -159.990, Y  +614.683, Z    +0.000, E1   +63.997, E3 -220451.304}
SPL {X  -159.990, Y  +629.274, Z    +0.000, E1   +64.033, E3 -220466.335}
SPL {X  -159.990, Y  +645.396, Z    +0.000, E1   +64.010, E3 -220483.066}
SPL {X  -159.990, Y  +656.294, Z    +0.000, E1   +63.988, E3 -220494.396}
SPL {X  -159.990, Y  +667.666, Z    +0.000, E1   +64.016, E3 -220506.087}
SPL {X  -159.767, Y  +679.937, Z    +0.000, E1   +63.968, E3 -220519.063}
SPL {X  -158.736, Y  +691.491, Z    +0.000, E1   +63.843, E3 -220532.061}
SPL {X  -157.131, Y  +701.612, Z    +0.000, E1   +63.591, E3 -220544.251}
SPL {X  -155.594, Y  +708.746, Z    +0.000, E1   +63.361, E3 -220553.231}
SPL {X  -153.286, Y  +717.329, Z    +0.000, E1   +63.046, E3 -220564.440}
SPL {X  -150.953, Y  +724.510, Z    +0.000, E1   +62.654, E3 -220574.268}
SPL {X  -148.087, Y  +732.056, Z    +0.000, E1   +62.252, E3 -220584.850}
SPL {X  -144.667, Y  +739.825, Z    +0.000, E1   +61.658, E3 -220596.239}
SPL {X  -142.263, Y  +744.698, Z    +0.000, E1   +61.245, E3 -220603.554}
SPL {X  -139.956, Y  +749.019, Z    +0.000, E1   +60.852, E3 -220610.132}
SPL {X  -136.617, Y  +754.762, Z    +0.000, E1   +60.296, E3 -220618.986}
SPL {X  -132.995, Y  +760.433, Z    +0.000, E1   +59.601, E3 -220627.950}
SPL {X  -109.949, Y  +787.724, Z    +0.000, E1   +51.944, E3 -220720.511}
ENDSPLINE

SPLINE
SPL {X  -129.366, Y  +765.635, Z    +0.000, E1   +44.361, E3 -220830.253}
SPL {X  -144.719, Y  +739.715, Z    +0.000, E1   +37.620, E3 -220857.101}
SPL {X  -154.606, Y  +712.654, Z    +0.000, E1   +26.872, E3 -220870.321}
SPL {X  -158.229, Y  +695.175, Z    +0.000, E1   +17.621, E3 -220874.807}
SPL {X  -159.735, Y  +680.532, Z    +0.000, E1    +8.352, E3 -220876.899}
SPL {X  -159.976, Y  +673.579, Z    +0.000, E1    +3.308, E3 -220877.393}
SPL {X  -159.990, Y  +669.438, Z    +0.000, E1    +0.061, E3 -220877.491}
SPL {X  -159.990, Y  +667.221, Z    +0.000, E1    -2.789, E3 -220877.534}
SPL {X  -159.990, Y  +663.611, Z    +0.000, E1    -7.967, E3 -220877.724}
SPL {X  -159.990, Y  +658.381, Z    +0.000, E1   -16.786, E3 -220878.205}
SPL {X  -159.990, Y  +651.878, Z    +0.000, E1   -27.298, E3 -220879.204}
SPL {X  -159.990, Y  +644.587, Z    +0.000, E1   -37.284, E3 -220880.787}
SPL {X  -159.990, Y  +633.621, Z    +0.000, E1   -47.309, E3 -220884.278}
SPL {X  -159.990, Y  +588.658, Z    +0.000, E1   -60.812, E3 -220906.598}
SPL {X  -159.990, Y  +495.038, Z    +0.000, E1   -63.580, E3 -220981.834}
SPL {X  -159.990, Y  +483.848, Z    +0.000, E1   -63.590, E3 -220993.619}
SPL {X  -159.990, Y  +471.874, Z    +0.000, E1   -63.586, E3 -221006.245}
SPL {X  -159.990, Y  +461.079, Z    +0.000, E1   -63.579, E3 -221017.653}
SPL {X  -159.990, Y  +450.188, Z    +0.000, E1   -63.581, E3 -221029.144}
SPL {X  -159.990, Y  +442.553, Z    +0.000, E1   -63.337, E3 -221038.967}
ENDSPLINE

SPLINE
SPL {X  -159.990, Y  +465.419, Z    +0.000, E1   -58.181, E3 -221047.813}
ENDSPLINE

SPLINE
SPL {X  -159.990, Y  +455.003, Z    +0.000, E1   -58.788, E3 -221057.351}
SPL {X  -159.990, Y  +443.180, Z    +0.000, E1   -59.522, E3 -221067.389}
SPL {X  -159.990, Y  +431.227, Z    +0.000, E1   -60.120, E3 -221078.081}
SPL {X  -159.990, Y  +413.464, Z    +0.000, E1   -61.043, E3 -221093.071}
SPL {X  -159.990, Y  +395.417, Z    +0.000, E1   -62.063, E3 -221106.514}
SPL {X  -159.983, Y  +381.042, Z    +0.000, E1   -62.802, E3 -221117.145}
SPL {X  -159.542, Y  +370.537, Z    +0.000, E1   -63.069, E3 -221126.527}
SPL {X  -158.758, Y  +362.683, Z    +0.000, E1   -62.956, E3 -221135.801}
SPL {X  -157.125, Y  +352.357, Z    +0.000, E1   -62.751, E3 -221148.534}
SPL {X  -154.421, Y  +340.656, Z    +0.000, E1   -62.344, E3 -221163.888}
SPL {X  -151.938, Y  +332.383, Z    +0.000, E1   -61.927, E3 -221175.360}
SPL {X  -149.604, Y  +325.796, Z    +0.000, E1   -61.568, E3 -221184.746}
SPL {X  -147.413, Y  +320.320, Z    +0.000, E1   -61.198, E3 -221192.799}
SPL {X  -145.235, Y  +315.391, Z    +0.000, E1   -60.847, E3 -221200.174}
SPL {X  -141.610, Y  +308.046, Z    +0.000, E1   -60.266, E3 -221211.410}
SPL {X  -138.010, Y  +301.568, Z    +0.000, E1   -59.585, E3 -221221.682}
SPL {X  -134.884, Y  +296.459, Z    +0.000, E1   -59.021, E3 -221229.863}
SPL {X  -132.471, Y  +292.789, Z    +0.000, E1   -58.532, E3 -221235.855}
SPL {X  -113.391, Y  +269.632, Z    +0.000, E1   -50.631, E3 -221330.903}
ENDSPLINE

SPLINE
SPL {X  -117.172, Y  +273.562, Z    +0.000, E1   -47.526, E3 -221379.054}
SPL {X  -141.985, Y  +308.763, Z    +0.000, E1   -38.695, E3 -221446.364}
SPL {X  -151.595, Y  +331.355, Z    +0.000, E1   -30.702, E3 -221460.883}
SPL {X  -155.358, Y  +344.279, Z    +0.000, E1   -24.937, E3 -221466.071}
SPL {X  -158.582, Y  +361.322, Z    +0.000, E1   -15.773, E3 -221470.415}
SPL {X  -159.657, Y  +372.183, Z    +0.000, E1    -8.995, E3 -221472.023}
SPL {X  -159.949, Y  +378.873, Z    +0.000, E1    -4.398, E3 -221472.598}
SPL {X  -159.990, Y  +382.801, Z    +0.000, E1    -1.461, E3 -221472.771}
SPL {X  -159.990, Y  +385.055, Z    +0.000, E1    +0.429, E3 -221472.811}
SPL {X  -159.990, Y  +388.743, Z    +0.000, E1    +5.147, E3 -221472.951}
SPL {X  -159.990, Y  +394.848, Z    +0.000, E1   +14.441, E3 -221473.491}
SPL {X  -159.990, Y  +402.771, Z    +0.000, E1   +27.045, E3 -221474.743}
SPL {X  -159.990, Y  +416.096, Z    +0.000, E1   +42.325, E3 -221478.411}
SPL {X  -159.990, Y  +469.763, Z    +0.000, E1   +60.937, E3 -221503.641}
SPL {X  -159.990, Y  +565.969, Z    +0.000, E1   +64.023, E3 -221579.414}
SPL {X  -159.990, Y  +578.082, Z    +0.000, E1   +63.987, E3 -221592.023}
SPL {X  -159.990, Y  +588.139, Z    +0.000, E1   +64.000, E3 -221602.403}
SPL {X  -159.990, Y  +601.786, Z    +0.000, E1   +64.016, E3 -221616.507}
SPL {X  -159.990, Y  +618.770, Z    +0.000, E1   +64.031, E3 -221634.043}
SPL {X  -159.990, Y  +636.111, Z    +0.000, E1   +64.024, E3 -221651.998}
SPL {X  -159.990, Y  +652.385, Z    +0.000, E1   +64.020, E3 -221668.855}
SPL {X  -159.990, Y  +667.666, Z    +0.000, E1   +64.016, E3 -221684.659}
SPL {X  -159.767, Y  +679.937, Z    +0.000, E1   +63.968, E3 -221697.634}
SPL {X  -159.113, Y  +688.225, Z    +0.000, E1   +63.867, E3 -221706.912}
SPL {X  -158.361, Y  +694.273, Z    +0.000, E1   +63.762, E3 -221713.950}
SPL {X  -157.131, Y  +701.612, Z    +0.000, E1   +63.591, E3 -221722.823}
SPL {X  -154.918, Y  +711.464, Z    +0.000, E1   +63.294, E3 -221735.258}
SPL {X  -152.656, Y  +719.385, Z    +0.000, E1   +62.921, E3 -221745.826}
SPL {X  -150.233, Y  +726.516, Z    +0.000, E1   +62.565, E3 -221755.604}
SPL {X  -147.385, Y  +733.745, Z    +0.000, E1   +62.104, E3 -221765.908}
SPL {X  -144.667, Y  +739.825, Z    +0.000, E1   +61.658, E3 -221774.811}
SPL {X  -142.263, Y  +744.698, Z    +0.000, E1   +61.245, E3 -221782.126}
SPL {X  -139.956, Y  +749.019, Z    +0.000, E1   +60.852, E3 -221788.703}
SPL {X  -136.617, Y  +754.762, Z    +0.000, E1   +60.296, E3 -221797.557}
SPL {X  -132.995, Y  +760.433, Z    +0.000, E1   +59.601, E3 -221806.521}
SPL {X  -109.949, Y  +787.724, Z    +0.000, E1   +51.944, E3 -221899.083}
ENDSPLINE

SPLINE
SPL {X  -129.366, Y  +765.635, Z    +0.000, E1   +44.361, E3 -222008.825}
SPL {X  -144.719, Y  +739.715, Z    +0.000, E1   +37.620, E3 -222035.672}
SPL {X  -154.606, Y  +712.654, Z    +0.000, E1   +26.872, E3 -222048.892}
SPL {X  -158.229, Y  +695.175, Z    +0.000, E1   +17.621, E3 -222053.378}
SPL {X  -159.735, Y  +680.532, Z    +0.000, E1    +8.352, E3 -222055.470}
SPL {X  -159.990, Y  +671.731, Z    +0.000, E1    +1.953, E3 -222056.020}
SPL {X  -159.990, Y  +669.188, Z    +0.000, E1    -0.261, E3 -222056.065}
SPL {X  -159.990, Y  +666.135, Z    +0.000, E1    -4.178, E3 -222056.154}
SPL {X  -159.990, Y  +662.249, Z    +0.000, E1   -10.338, E3 -222056.385}
SPL {X  -159.990, Y  +658.381, Z    +0.000, E1   -16.786, E3 -222056.777}
SPL {X  -159.990, Y  +651.878, Z    +0.000, E1   -27.298, E3 -222057.776}
SPL {X  -159.990, Y  +644.587, Z    +0.000, E1   -37.284, E3 -222059.358}
SPL {X  -159.990, Y  +633.621, Z    +0.000, E1   -47.309, E3 -222062.849}
SPL {X  -159.990, Y  +588.658, Z    +0.000, E1   -60.812, E3 -222085.169}
SPL {X  -159.990, Y  +495.038, Z    +0.000, E1   -63.580, E3 -222160.406}
SPL {X  -159.990, Y  +483.848, Z    +0.000, E1   -63.590, E3 -222172.190}
SPL {X  -159.990, Y  +471.874, Z    +0.000, E1   -63.586, E3 -222184.816}
SPL {X  -159.990, Y  +461.079, Z    +0.000, E1   -63.579, E3 -222196.225}
SPL {X  -159.990, Y  +450.188, Z    +0.000, E1   -63.581, E3 -222207.715}
SPL {X  -159.990, Y  +442.553, Z    +0.000, E1   -63.337, E3 -222217.539}
ENDSPLINE

SPLINE
SPL {X  -159.990, Y  +465.419, Z    +0.000, E1   -58.181, E3 -222226.384}
ENDSPLINE

SPLINE
SPL {X  -159.990, Y  +455.003, Z    +0.000, E1   -58.788, E3 -222235.922}
SPL {X  -159.990, Y  +443.180, Z    +0.000, E1   -59.522, E3 -222245.961}
SPL {X  -159.990, Y  +431.227, Z    +0.000, E1   -60.120, E3 -222256.653}
SPL {X  -159.990, Y  +413.464, Z    +0.000, E1   -61.043, E3 -222271.643}
SPL {X  -159.990, Y  +395.417, Z    +0.000, E1   -62.063, E3 -222285.086}
SPL {X  -159.983, Y  +381.042, Z    +0.000, E1   -62.802, E3 -222295.717}
SPL {X  -159.542, Y  +370.537, Z    +0.000, E1   -63.069, E3 -222305.099}
SPL {X  -158.758, Y  +362.683, Z    +0.000, E1   -62.956, E3 -222314.373}
SPL {X  -157.125, Y  +352.357, Z    +0.000, E1   -62.751, E3 -222327.106}
SPL {X  -155.132, Y  +343.375, Z    +0.000, E1   -62.418, E3 -222338.865}
SPL {X  -152.656, Y  +334.615, Z    +0.000, E1   -62.078, E3 -222350.742}
SPL {X  -149.604, Y  +325.796, Z    +0.000, E1   -61.568, E3 -222363.318}
SPL {X  -147.413, Y  +320.320, Z    +0.000, E1   -61.198, E3 -222371.371}
SPL {X  -145.235, Y  +315.391, Z    +0.000, E1   -60.847, E3 -222378.746}
SPL {X  -142.998, Y  +310.747, Z    +0.000, E1   -60.455, E3 -222385.858}
SPL {X  -140.747, Y  +306.427, Z    +0.000, E1   -60.074, E3 -222392.567}
SPL {X  -138.010, Y  +301.568, Z    +0.000, E1   -59.585, E3 -222400.253}
SPL {X  -134.884, Y  +296.459, Z    +0.000, E1   -59.021, E3 -222408.434}
SPL {X  -132.471, Y  +292.789, Z    +0.000, E1   -58.532, E3 -222414.426}
SPL {X  -113.541, Y  +269.782, Z    +0.000, E1   -50.113, E3 -222516.983}
ENDSPLINE

SPLINE
SPL {X  -145.506, Y  +315.982, Z    +0.000, E1   -36.457, E3 -222630.218}
SPL {X  -155.358, Y  +344.279, Z    +0.000, E1   -24.937, E3 -222644.643}
SPL {X  -158.582, Y  +361.322, Z    +0.000, E1   -15.773, E3 -222648.987}
SPL {X  -159.657, Y  +372.183, Z    +0.000, E1    -8.995, E3 -222650.595}
SPL {X  -159.949, Y  +378.873, Z    +0.000, E1    -4.398, E3 -222651.169}
SPL {X  -159.990, Y  +382.801, Z    +0.000, E1    -1.461, E3 -222651.343}
SPL {X  -159.990, Y  +384.517, Z    +0.000, E1    -0.022, E3 -222651.373}
SPL {X  -159.990, Y  +386.497, Z    +0.000, E1    +2.123, E3 -222651.421}
SPL {X  -159.990, Y  +391.572, Z    +0.000, E1    +9.236, E3 -222651.727}
SPL {X  -159.990, Y  +397.198, Z    +0.000, E1   +18.490, E3 -222652.352}
SPL {X  -159.990, Y  +402.771, Z    +0.000, E1   +27.045, E3 -222653.315}
SPL {X  -159.990, Y  +410.571, Z    +0.000, E1   +37.149, E3 -222655.131}
SPL {X  -159.990, Y  +420.033, Z    +0.000, E1   +45.596, E3 -222658.297}
SPL {X  -159.990, Y  +469.763, Z    +0.000, E1   +60.937, E3 -222682.212}
SPL {X  -159.990, Y  +561.242, Z    +0.000, E1   +63.988, E3 -222753.160}
SPL {X  -159.990, Y  +574.019, Z    +0.000, E1   +64.020, E3 -222766.326}
SPL {X  -159.990, Y  +591.720, Z    +0.000, E1   +64.032, E3 -222784.625}
SPL {X  -159.990, Y  +605.088, Z    +0.000, E1   +63.988, E3 -222798.552}
SPL {X  -159.990, Y  +614.683, Z    +0.000, E1   +63.997, E3 -222808.447}
SPL {X  -159.990, Y  +629.274, Z    +0.000, E1   +64.033, E3 -222823.478}
SPL {X  -159.990, Y  +645.396, Z    +0.000, E1   +64.010, E3 -222840.209}
SPL {X  -159.990, Y  +659.675, Z    +0.000, E1   +64.013, E3 -222854.981}
SPL {X  -159.990, Y  +670.719, Z    +0.000, E1   +63.993, E3 -222866.430}
SPL {X  -159.767, Y  +679.937, Z    +0.000, E1   +63.968, E3 -222876.206}
SPL {X  -158.736, Y  +691.491, Z    +0.000, E1   +63.843, E3 -222889.204}
SPL {X  -157.131, Y  +701.612, Z    +0.000, E1   +63.591, E3 -222901.394}
SPL {X  -154.918, Y  +711.464, Z    +0.000, E1   +63.294, E3 -222913.829}
SPL {X  -151.874, Y  +721.810, Z    +0.000, E1   +62.834, E3 -222927.636}
SPL {X  -148.087, Y  +732.056, Z    +0.000, E1   +62.252, E3 -222941.993}
SPL {X  -144.667, Y  +739.825, Z    +0.000, E1   +61.658, E3 -222953.382}
SPL {X  -142.263, Y  +744.698, Z    +0.000, E1   +61.245, E3 -222960.697}
SPL {X  -138.935, Y  +750.833, Z    +0.000, E1   +60.711, E3 -222970.022}
SPL {X  -135.668, Y  +756.300, Z    +0.000, E1   +60.086, E3 -222978.585}
SPL {X  -132.995, Y  +760.433, Z    +0.000, E1   +59.601, E3 -222985.093}
SPL {X  -109.949, Y  +787.724, Z    +0.000, E1   +51.944, E3 -223077.654}
ENDSPLINE

SPLINE
SPL {X  -129.366, Y  +765.635, Z    +0.000, E1   +44.361, E3 -223187.396}
SPL {X  -144.719, Y  +739.715, Z    +0.000, E1   +37.620, E3 -223214.244}
SPL {X  -154.606, Y  +712.654, Z    +0.000, E1   +26.872, E3 -223227.464}
SPL {X  -158.229, Y  +695.175, Z    +0.000, E1   +17.621, E3 -223231.950}
SPL {X  -159.735, Y  +680.532, Z    +0.000, E1    +8.352, E3 -223234.042}
SPL {X  -159.990, Y  +671.731, Z    +0.000, E1    +1.953, E3 -223234.592}
SPL {X  -159.990, Y  +669.188, Z    +0.000, E1    -0.261, E3 -223234.636}
SPL {X  -159.990, Y  +666.135, Z    +0.000, E1    -4.178, E3 -223234.725}
SPL {X  -159.990, Y  +662.249, Z    +0.000, E1   -10.338, E3 -223234.956}
SPL {X  -159.990, Y  +658.381, Z    +0.000, E1   -16.786, E3 -223235.348}
SPL {X  -159.990, Y  +651.878, Z    +0.000, E1   -27.298, E3 -223236.347}
SPL {X  -159.990, Y  +644.587, Z    +0.000, E1   -37.284, E3 -223237.930}
SPL {X  -159.990, Y  +633.621, Z    +0.000, E1   -47.309, E3 -223241.421}
SPL {X  -159.990, Y  +588.658, Z    +0.000, E1   -60.812, E3 -223263.741}
SPL {X  -159.990, Y  +495.038, Z    +0.000, E1   -63.580, E3 -223338.977}
SPL {X  -159.990, Y  +483.848, Z    +0.000, E1   -63.590, E3 -223350.762}
SPL {X  -159.990, Y  +471.874, Z    +0.000, E1   -63.586, E3 -223363.387}
SPL {X  -159.990, Y  +461.079, Z    +0.000, E1   -63.579, E3 -223374.796}
SPL {X  -159.990, Y  +450.188, Z    +0.000, E1   -63.581, E3 -223386.287}
SPL {X  -159.990, Y  +442.553, Z    +0.000, E1   -63.337, E3 -223396.110}
ENDSPLINE

SPLINE
SPL {X  -159.990, Y  +465.419, Z    +0.000, E1   -58.181, E3 -223404.956}
ENDSPLINE

SPLINE
SPL {X  -159.990, Y  +455.003, Z    +0.000, E1   -58.788, E3 -223414.494}
SPL {X  -159.990, Y  +443.180, Z    +0.000, E1   -59.522, E3 -223424.532}
SPL {X  -159.990, Y  +431.227, Z    +0.000, E1   -60.120, E3 -223435.224}
SPL {X  -159.990, Y  +413.464, Z    +0.000, E1   -61.043, E3 -223450.214}
SPL {X  -159.990, Y  +395.417, Z    +0.000, E1   -62.063, E3 -223463.657}
SPL {X  -159.983, Y  +381.042, Z    +0.000, E1   -62.802, E3 -223474.288}
SPL {X  -159.542, Y  +370.537, Z    +0.000, E1   -63.069, E3 -223483.670}
SPL {X  -158.758, Y  +362.683, Z    +0.000, E1   -62.956, E3 -223492.944}
SPL {X  -157.125, Y  +352.357, Z    +0.000, E1   -62.751, E3 -223505.677}
SPL {X  -154.421, Y  +340.656, Z    +0.000, E1   -62.344, E3 -223521.031}
SPL {X  -151.938, Y  +332.383, Z    +0.000, E1   -61.927, E3 -223532.503}
SPL {X  -149.604, Y  +325.796, Z    +0.000, E1   -61.568, E3 -223541.889}
SPL {X  -147.413, Y  +320.320, Z    +0.000, E1   -61.198, E3 -223549.942}
SPL {X  -145.235, Y  +315.391, Z    +0.000, E1   -60.847, E3 -223557.317}
SPL {X  -141.610, Y  +308.046, Z    +0.000, E1   -60.266, E3 -223568.553}
SPL {X  -138.010, Y  +301.568, Z    +0.000, E1   -59.585, E3 -223578.825}
SPL {X  -134.884, Y  +296.459, Z    +0.000, E1   -59.021, E3 -223587.006}
SPL {X  -132.471, Y  +292.789, Z    +0.000, E1   -58.532, E3 -223592.998}
SPL {X  -113.391, Y  +269.632, Z    +0.000, E1   -50.631, E3 -223688.046}
ENDSPLINE

SPLINE
SPL {X  -117.172, Y  +273.562, Z    +0.000, E1   -47.526, E3 -223736.197}
SPL {X  -141.985, Y  +308.763, Z    +0.000, E1   -38.695, E3 -223803.507}
SPL {X  -151.595, Y  +331.355, Z    +0.000, E1   -30.702, E3 -223818.026}
SPL {X  -155.358, Y  +344.279, Z    +0.000, E1   -24.937, E3 -223823.214}
SPL {X  -158.582, Y  +361.322, Z    +0.000, E1   -15.773, E3 -223827.558}
SPL {X  -159.657, Y  +372.183, Z    +0.000, E1    -8.995, E3 -223829.166}
SPL {X  -159.949, Y  +378.873, Z    +0.000, E1    -4.398, E3 -223829.740}
SPL {X  -159.990, Y  +382.801, Z    +0.000, E1    -1.461, E3 -223829.914}
SPL {X  -159.990, Y  +385.055, Z    +0.000, E1    +0.429, E3 -223829.953}
SPL {X  -159.990, Y  +388.743, Z    +0.000, E1    +5.147, E3 -223830.094}
SPL {X  -159.990, Y  +394.848, Z    +0.000, E1   +14.441, E3 -223830.634}
SPL {X  -159.990, Y  +402.771, Z    +0.000, E1   +27.045, E3 -223831.886}
SPL {X  -159.990, Y  +416.096, Z    +0.000, E1   +42.325, E3 -223835.554}
SPL {X  -159.990, Y  +469.763, Z    +0.000, E1   +60.937, E3 -223860.783}
SPL {X  -159.990, Y  +561.242, Z    +0.000, E1   +63.988, E3 -223931.732}
SPL {X  -159.990, Y  +574.019, Z    +0.000, E1   +64.020, E3 -223944.898}
SPL {X  -159.990, Y  +591.720, Z    +0.000, E1   +64.032, E3 -223963.196}
SPL {X  -159.990, Y  +605.088, Z    +0.000, E1   +63.988, E3 -223977.124}
SPL {X  -159.990, Y  +614.683, Z    +0.000, E1   +63.997, E3 -223987.018}
SPL {X  -159.990, Y  +629.274, Z    +0.000, E1   +64.033, E3 -224002.049}
SPL {X  -159.990, Y  +645.396, Z    +0.000, E1   +64.010, E3 -224018.780}
SPL {X  -159.990, Y  +656.294, Z    +0.000, E1   +63.988, E3 -224030.110}
SPL {X  -159.990, Y  +667.666, Z    +0.000, E1   +64.016, E3 -224041.802}
SPL {X  -159.767, Y  +679.937, Z    +0.000, E1   +63.968, E3 -224054.777}
SPL {X  -159.113, Y  +688.225, Z    +0.000, E1   +63.867, E3 -224064.055}
SPL {X  -158.361, Y  +694.273, Z    +0.000, E1   +63.762, E3 -224071.092}
SPL {X  -157.131, Y  +701.612, Z    +0.000, E1   +63.591, E3 -224079.965}
SPL {X  -154.918, Y  +711.464, Z    +0.000, E1   +63.294, E3 -224092.401}
SPL {X  -151.874, Y  +721.810, Z    +0.000, E1   +62.834, E3 -224106.207}
SPL {X  -148.087, Y  +732.056, Z    +0.000, E1   +62.252, E3 -224120.564}
SPL {X  -144.667, Y  +739.825, Z    +0.000, E1   +61.658, E3 -224131.953}
SPL {X  -142.263, Y  +744.698, Z    +0.000, E1   +61.245, E3 -224139.269}
SPL {X  -138.935, Y  +750.833, Z    +0.000, E1   +60.711, E3 -224148.593}
SPL {X  -135.668, Y  +756.300, Z    +0.000, E1   +60.086, E3 -224157.156}
SPL {X  -132.995, Y  +760.433, Z    +0.000, E1   +59.601, E3 -224163.664}
SPL {X  -109.949, Y  +787.724, Z    +0.000, E1   +51.944, E3 -224256.226}
ENDSPLINE

SPLINE
SPL {X  -129.366, Y  +765.635, Z    +0.000, E1   +44.361, E3 -224365.968}
SPL {X  -144.719, Y  +739.715, Z    +0.000, E1   +37.620, E3 -224392.815}
SPL {X  -154.606, Y  +712.654, Z    +0.000, E1   +26.872, E3 -224406.035}
SPL {X  -158.229, Y  +695.175, Z    +0.000, E1   +17.621, E3 -224410.521}
SPL {X  -159.735, Y  +680.532, Z    +0.000, E1    +8.352, E3 -224412.613}
SPL {X  -159.990, Y  +671.731, Z    +0.000, E1    +1.953, E3 -224413.163}
SPL {X  -159.990, Y  +668.624, Z    +0.000, E1    -0.752, E3 -224413.219}
SPL {X  -159.990, Y  +663.611, Z    +0.000, E1    -7.967, E3 -224413.439}
SPL {X  -159.990, Y  +658.381, Z    +0.000, E1   -16.786, E3 -224413.919}
SPL {X  -159.990, Y  +651.878, Z    +0.000, E1   -27.298, E3 -224414.918}
SPL {X  -159.990, Y  +644.587, Z    +0.000, E1   -37.284, E3 -224416.501}
SPL {X  -159.990, Y  +633.621, Z    +0.000, E1   -47.309, E3 -224419.992}
SPL {X  -159.990, Y  +588.658, Z    +0.000, E1   -60.812, E3 -224442.312}
SPL {X  -159.990, Y  +495.038, Z    +0.000, E1   -63.580, E3 -224517.548}
SPL {X  -159.990, Y  +483.848, Z    +0.000, E1   -63.590, E3 -224529.333}
SPL {X  -159.990, Y  +471.874, Z    +0.000, E1   -63.586, E3 -224541.959}
SPL {X  -159.990, Y  +461.079, Z    +0.000, E1   -63.579, E3 -224553.367}
SPL {X  -159.990, Y  +450.188, Z    +0.000, E1   -63.581, E3 -224564.858}
SPL {X  -159.990, Y  +442.553, Z    +0.000, E1   -63.337, E3 -224574.682}
ENDSPLINE

SPLINE
SPL {X  -159.990, Y  +465.419, Z    +0.000, E1   -58.181, E3 -224583.527}
ENDSPLINE

SPLINE
SPL {X  -159.990, Y  +455.003, Z    +0.000, E1   -58.788, E3 -224593.065}
SPL {X  -159.990, Y  +443.180, Z    +0.000, E1   -59.522, E3 -224603.103}
SPL {X  -159.990, Y  +431.227, Z    +0.000, E1   -60.120, E3 -224613.796}
SPL {X  -159.990, Y  +413.464, Z    +0.000, E1   -61.043, E3 -224628.786}
SPL {X  -159.990, Y  +395.417, Z    +0.000, E1   -62.063, E3 -224642.228}
SPL {X  -159.983, Y  +381.042, Z    +0.000, E1   -62.802, E3 -224652.860}
SPL {X  -159.542, Y  +370.537, Z    +0.000, E1   -63.069, E3 -224662.242}
SPL {X  -158.758, Y  +362.683, Z    +0.000, E1   -62.956, E3 -224671.515}
SPL {X  -157.125, Y  +352.357, Z    +0.000, E1   -62.751, E3 -224684.249}
SPL {X  -154.421, Y  +340.656, Z    +0.000, E1   -62.344, E3 -224699.602}
SPL {X  -151.938, Y  +332.383, Z    +0.000, E1   -61.927, E3 -224711.075}
SPL {X  -149.604, Y  +325.796, Z    +0.000, E1   -61.568, E3 -224720.461}
SPL {X  -147.413, Y  +320.320, Z    +0.000, E1   -61.198, E3 -224728.514}
SPL {X  -145.235, Y  +315.391, Z    +0.000, E1   -60.847, E3 -224735.888}
SPL {X  -141.610, Y  +308.046, Z    +0.000, E1   -60.266, E3 -224747.125}
SPL {X  -137.263, Y  +300.308, Z    +0.000, E1   -59.477, E3 -224759.374}
SPL {X  -133.767, Y  +294.732, Z    +0.000, E1   -58.799, E3 -224768.382}
SPL {X  -113.541, Y  +269.782, Z    +0.000, E1   -50.113, E3 -224874.126}
ENDSPLINE

SPLINE
SPL {X  -145.506, Y  +315.982, Z    +0.000, E1   -36.457, E3 -224987.361}
SPL {X  -155.358, Y  +344.279, Z    +0.000, E1   -24.937, E3 -225001.786}
SPL {X  -158.582, Y  +361.322, Z    +0.000, E1   -15.773, E3 -225006.129}
SPL {X  -159.657, Y  +372.183, Z    +0.000, E1    -8.995, E3 -225007.738}
SPL {X  -159.949, Y  +378.873, Z    +0.000, E1    -4.398, E3 -225008.312}
SPL {X  -159.990, Y  +382.801, Z    +0.000, E1    -1.461, E3 -225008.485}
SPL {X  -159.990, Y  +385.055, Z    +0.000, E1    +0.429, E3 -225008.525}
SPL {X  -159.990, Y  +388.743, Z    +0.000, E1    +5.147, E3 -225008.666}
SPL {X  -159.990, Y  +393.154, Z    +0.000, E1   +11.942, E3 -225008.997}
SPL {X  -159.990, Y  +397.198, Z    +0.000, E1   +18.490, E3 -225009.494}
SPL {X  -159.990, Y  +402.771, Z    +0.000, E1   +27.045, E3 -225010.458}
SPL {X  -159.990, Y  +416.096, Z    +0.000, E1   +42.325, E3 -225014.125}
SPL {X  -159.990, Y  +469.763, Z    +0.000, E1   +60.937, E3 -225039.355}
SPL {X  -159.990, Y  +561.242, Z    +0.000, E1   +63.988, E3 -225110.303}
SPL {X  -159.990, Y  +574.019, Z    +0.000, E1   +64.020, E3 -225123.469}
SPL {X  -159.990, Y  +591.720, Z    +0.000, E1   +64.032, E3 -225141.768}
SPL {X  -159.990, Y  +605.088, Z    +0.000, E1   +63.988, E3 -225155.695}
SPL {X  -159.990, Y  +614.683, Z    +0.000, E1   +63.997, E3 -225165.590}
SPL {X  -159.990, Y  +629.274, Z    +0.000, E1   +64.033, E3 -225180.621}
SPL {X  -159.990, Y  +645.396, Z    +0.000, E1   +64.010, E3 -225197.352}
SPL {X  -159.990, Y  +656.294, Z    +0.000, E1   +63.988, E3 -225208.681}
SPL {X  -159.990, Y  +667.666, Z    +0.000, E1   +64.016, E3 -225220.373}
SPL {X  -159.767, Y  +679.937, Z    +0.000, E1   +63.968, E3 -225233.348}
SPL {X  -158.736, Y  +691.491, Z    +0.000, E1   +63.843, E3 -225246.347}
SPL {X  -157.131, Y  +701.612, Z    +0.000, E1   +63.591, E3 -225258.537}
SPL {X  -155.594, Y  +708.746, Z    +0.000, E1   +63.361, E3 -225267.517}
SPL {X  -153.286, Y  +717.329, Z    +0.000, E1   +63.046, E3 -225278.725}
SPL {X  -150.953, Y  +724.510, Z    +0.000, E1   +62.654, E3 -225288.553}
SPL {X  -148.087, Y  +732.056, Z    +0.000, E1   +62.252, E3 -225299.135}
SPL {X  -144.667, Y  +739.825, Z    +0.000, E1   +61.658, E3 -225310.525}
SPL {X  -142.263, Y  +744.698, Z    +0.000, E1   +61.245, E3 -225317.840}
SPL {X  -138.935, Y  +750.833, Z    +0.000, E1   +60.711, E3 -225327.165}
SPL {X  -135.668, Y  +756.300, Z    +0.000, E1   +60.086, E3 -225335.728}
SPL {X  -132.995, Y  +760.433, Z    +0.000, E1   +59.601, E3 -225342.235}
SPL {X  -109.949, Y  +787.724, Z    +0.000, E1   +51.944, E3 -225434.797}
ENDSPLINE

SPLINE
SPL {X  -129.366, Y  +765.635, Z    +0.000, E1   +44.361, E3 -225544.539}
SPL {X  -144.719, Y  +739.715, Z    +0.000, E1   +37.620, E3 -225571.386}
SPL {X  -154.606, Y  +712.654, Z    +0.000, E1   +26.872, E3 -225584.606}
SPL {X  -158.229, Y  +695.175, Z    +0.000, E1   +17.621, E3 -225589.092}
SPL {X  -159.536, Y  +683.548, Z    +0.000, E1   +10.326, E3 -225590.880}
SPL {X  -159.946, Y  +675.243, Z    +0.000, E1    +4.608, E3 -225591.589}
SPL {X  -159.990, Y  +670.644, Z    +0.000, E1    +1.007, E3 -225591.764}
SPL {X  -159.990, Y  +669.188, Z    +0.000, E1    -0.261, E3 -225591.779}
SPL {X  -159.990, Y  +666.135, Z    +0.000, E1    -4.178, E3 -225591.868}
SPL {X  -159.990, Y  +662.249, Z    +0.000, E1   -10.338, E3 -225592.099}
SPL {X  -159.990, Y  +658.381, Z    +0.000, E1   -16.786, E3 -225592.491}
SPL {X  -159.990, Y  +651.878, Z    +0.000, E1   -27.298, E3 -225593.490}
SPL {X  -159.990, Y  +644.587, Z    +0.000, E1   -37.284, E3 -225595.073}
SPL {X  -159.990, Y  +633.621, Z    +0.000, E1   -47.309, E3 -225598.564}
SPL {X  -159.990, Y  +588.658, Z    +0.000, E1   -60.812, E3 -225620.884}
SPL {X  -159.990, Y  +495.038, Z    +0.000, E1   -63.580, E3 -225696.120}
SPL {X  -159.990, Y  +483.848, Z    +0.000, E1   -63.590, E3 -225707.905}
SPL {X  -159.990, Y  +471.874, Z    +0.000, E1   -63.586, E3 -225720.530}
SPL {X  -159.990, Y  +461.079, Z    +0.000, E1   -63.579, E3 -225731.939}
SPL {X  -159.990, Y  +450.188, Z    +0.000, E1   -63.581, E3 -225743.429}
SPL {X  -159.990, Y  +442.553, Z    +0.000, E1   -63.337, E3 -225753.253}
ENDSPLINE

SPLINE
SPL {X  -159.990, Y  +465.419, Z    +0.000, E1   -58.181, E3 -225762.098}
ENDSPLINE

SPLINE
SPL {X  -159.990, Y  +455.003, Z    +0.000, E1   -58.788, E3 -225771.637}
SPL {X  -159.990, Y  +443.180, Z    +0.000, E1   -59.522, E3 -225781.675}
SPL {X  -159.990, Y  +431.227, Z    +0.000, E1   -60.120, E3 -225792.367}
SPL {X  -159.990, Y  +413.464, Z    +0.000, E1   -61.043, E3 -225807.357}
SPL {X  -159.990, Y  +395.417, Z    +0.000, E1   -62.063, E3 -225820.800}
SPL {X  -159.983, Y  +381.042, Z    +0.000, E1   -62.802, E3 -225831.431}
SPL {X  -159.542, Y  +370.537, Z    +0.000, E1   -63.069, E3 -225840.813}
SPL {X  -158.287, Y  +359.218, Z    +0.000, E1   -62.927, E3 -225854.228}
SPL {X  -155.813, Y  +346.180, Z    +0.000, E1   -62.560, E3 -225870.805}
SPL {X  -152.656, Y  +334.615, Z    +0.000, E1   -62.078, E3 -225886.457}
SPL {X  -149.604, Y  +325.796, Z    +0.000, E1   -61.568, E3 -225899.032}
SPL {X  -147.413, Y  +320.320, Z    +0.000, E1   -61.198, E3 -225907.085}
SPL {X  -145.235, Y  +315.391, Z    +0.000, E1   -60.847, E3 -225914.460}
SPL {X  -141.610, Y  +308.046, Z    +0.000, E1   -60.266, E3 -225925.696}
SPL {X  -137.263, Y  +300.308, Z    +0.000, E1   -59.477, E3 -225937.946}
SPL {X  -133.767, Y  +294.732, Z    +0.000, E1   -58.799, E3 -225946.954}
SPL {X  -113.541, Y  +269.782, Z    +0.000, E1   -50.113, E3 -226052.697}
ENDSPLINE

SPLINE
SPL {X  -141.985, Y  +308.763, Z    +0.000, E1   -38.695, E3 -226160.650}
SPL {X  -154.491, Y  +340.913, Z    +0.000, E1   -26.570, E3 -226179.102}
SPL {X  -158.582, Y  +361.322, Z    +0.000, E1   -15.773, E3 -226184.701}
SPL {X  -159.657, Y  +372.183, Z    +0.000, E1    -8.995, E3 -226186.309}
SPL {X  -159.986, Y  +381.348, Z    +0.000, E1    -2.678, E3 -226186.998}
SPL {X  -159.990, Y  +384.517, Z    +0.000, E1    -0.022, E3 -226187.087}
SPL {X  -159.990, Y  +386.497, Z    +0.000, E1    +2.123, E3 -226187.135}
SPL {X  -159.990, Y  +391.572, Z    +0.000, E1    +9.236, E3 -226187.441}
SPL {X  -159.990, Y  +397.198, Z    +0.000, E1   +18.490, E3 -226188.066}
SPL {X  -159.990, Y  +402.771, Z    +0.000, E1   +27.045, E3 -226189.029}
SPL {X  -159.990, Y  +414.719, Z    +0.000, E1   +41.161, E3 -226192.203}
SPL {X  -159.990, Y  +424.336, Z    +0.000, E1   +48.481, E3 -226195.638}
SPL {X  -159.990, Y  +469.763, Z    +0.000, E1   +60.937, E3 -226217.926}
SPL {X  -159.990, Y  +561.242, Z    +0.000, E1   +63.988, E3 -226288.875}
SPL {X  -159.990, Y  +574.019, Z    +0.000, E1   +64.020, E3 -226302.041}
SPL {X  -159.990, Y  +591.720, Z    +0.000, E1   +64.032, E3 -226320.339}
SPL {X  -159.990, Y  +605.088, Z    +0.000, E1   +63.988, E3 -226334.266}
SPL {X  -159.990, Y  +614.683, Z    +0.000, E1   +63.997, E3 -226344.161}
SPL {X  -159.990, Y  +629.274, Z    +0.000, E1   +64.033, E3 -226359.192}
SPL {X  -159.990, Y  +645.396, Z    +0.000, E1   +64.010, E3 -226375.923}
SPL {X  -159.990, Y  +659.675, Z    +0.000, E1   +64.013, E3 -226390.695}
SPL {X  -159.990, Y  +670.719, Z    +0.000, E1   +63.993, E3 -226402.145}
SPL {X  -159.767, Y  +679.937, Z    +0.000, E1   +63.968, E3 -226411.920}
SPL {X  -158.736, Y  +691.491, Z    +0.000, E1   +63.843, E3 -226424.918}
SPL {X  -157.131, Y  +701.612, Z    +0.000, E1   +63.591, E3 -226437.108}
SPL {X  -155.594, Y  +708.746, Z    +0.000, E1   +63.361, E3 -226446.088}
SPL {X  -153.286, Y  +717.329, Z    +0.000, E1   +63.046, E3 -226457.297}
SPL {X  -150.233, Y  +726.516, Z    +0.000, E1   +62.565, E3 -226469.890}
SPL {X  -147.385, Y  +733.745, Z    +0.000, E1   +62.104, E3 -226480.194}
SPL {X  -144.667, Y  +739.825, Z    +0.000, E1   +61.658, E3 -226489.096}
SPL {X  -142.263, Y  +744.698, Z    +0.000, E1   +61.245, E3 -226496.412}
SPL {X  -139.956, Y  +749.019, Z    +0.000, E1   +60.852, E3 -226502.989}
SPL {X  -136.617, Y  +754.762, Z    +0.000, E1   +60.296, E3 -226511.843}
SPL {X  -132.995, Y  +760.433, Z    +0.000, E1   +59.601, E3 -226520.807}
SPL {X  -109.949, Y  +787.724, Z    +0.000, E1   +51.944, E3 -226613.368}
ENDSPLINE

SPLINE
SPL {X  -129.366, Y  +765.635, Z    +0.000, E1   +44.361, E3 -226723.110}
SPL {X  -144.719, Y  +739.715, Z    +0.000, E1   +37.620, E3 -226749.958}
SPL {X  -154.606, Y  +712.654, Z    +0.000, E1   +26.872, E3 -226763.178}
SPL {X  -158.229, Y  +695.175, Z    +0.000, E1   +17.621, E3 -226767.664}
SPL {X  -159.735, Y  +680.532, Z    +0.000, E1    +8.352, E3 -226769.756}
SPL {X  -159.990, Y  +671.731, Z    +0.000, E1    +1.953, E3 -226770.306}
SPL {X  -159.990, Y  +669.188, Z    +0.000, E1    -0.261, E3 -226770.351}
SPL {X  -159.990, Y  +666.135, Z    +0.000, E1    -4.178, E3 -226770.439}
SPL {X  -159.990, Y  +662.249, Z    +0.000, E1   -10.338, E3 -226770.671}
SPL {X  -159.990, Y  +658.381, Z    +0.000, E1   -16.786, E3 -226771.062}
SPL {X  -159.990, Y  +651.878, Z    +0.000, E1   -27.298, E3 -226772.061}
SPL {X  -159.990, Y  +644.587, Z    +0.000, E1   -37.284, E3 -226773.644}
SPL {X  -159.990, Y  +633.621, Z    +0.000, E1   -47.309, E3 -226777.135}
SPL {X  -159.990, Y  +588.658, Z    +0.000, E1   -60.812, E3 -226799.455}
SPL {X  -159.990, Y  +495.038, Z    +0.000, E1   -63.580, E3 -226874.691}
SPL {X  -159.990, Y  +483.848, Z    +0.000, E1   -63.590, E3 -226886.476}
SPL {X  -159.990, Y  +471.874, Z    +0.000, E1   -63.586, E3 -226899.102}
SPL {X  -159.990, Y  +461.079, Z    +0.000, E1   -63.579, E3 -226910.510}
SPL {X  -159.990, Y  +450.188, Z    +0.000, E1   -63.581, E3 -226922.001}
SPL {X  -159.990, Y  +442.553, Z    +0.000, E1   -63.337, E3 -226931.824}
ENDSPLINE

SPLINE
SPL {X  -159.990, Y  +465.419, Z    +0.000, E1   -58.181, E3 -226940.670}
ENDSPLINE

SPLINE
SPL {X  -159.990, Y  +455.003, Z    +0.000, E1   -58.788, E3 -226950.208}
SPL {X  -159.990, Y  +443.180, Z    +0.000, E1   -59.522, E3 -226960.246}
SPL {X  -159.990, Y  +431.227, Z    +0.000, E1   -60.120, E3 -226970.938}
SPL {X  -159.990, Y  +418.989, Z    +0.000, E1   -60.714, E3 -226981.574}
SPL {X  -159.990, Y  +401.382, Z    +0.000, E1   -61.735, E3 -226995.043}
SPL {X  -159.983, Y  +381.042, Z    +0.000, E1   -62.802, E3 -227010.003}
SPL {X  -159.542, Y  +370.537, Z    +0.000, E1   -63.069, E3 -227019.385}
SPL {X  -158.287, Y  +359.218, Z    +0.000, E1   -62.927, E3 -227032.799}
SPL {X  -155.813, Y  +346.180, Z    +0.000, E1   -62.560, E3 -227049.376}
SPL {X  -152.656, Y  +334.615, Z    +0.000, E1   -62.078, E3 -227065.028}
SPL {X  -149.604, Y  +325.796, Z    +0.000, E1   -61.568, E3 -227077.603}
SPL {X  -147.413, Y  +320.320, Z    +0.000, E1   -61.198, E3 -227085.657}
SPL {X  -145.235, Y  +315.391, Z    +0.000, E1   -60.847, E3 -227093.031}
SPL {X  -141.610, Y  +308.046, Z    +0.000, E1   -60.266, E3 -227104.268}
SPL {X  -138.010, Y  +301.568, Z    +0.000, E1   -59.585, E3 -227114.539}
SPL {X  -134.884, Y  +296.459, Z    +0.000, E1   -59.021, E3 -227122.720}
SPL {X  -132.471, Y  +292.789, Z    +0.000, E1   -58.532, E3 -227128.712}
SPL {X  -113.391, Y  +269.632, Z    +0.000, E1   -50.631, E3 -227223.760}
ENDSPLINE

SPLINE
SPL {X  -117.172, Y  +273.562, Z    +0.000, E1   -47.526, E3 -227271.911}
SPL {X  -141.985, Y  +308.763, Z    +0.000, E1   -38.695, E3 -227339.221}
SPL {X  -151.595, Y  +331.355, Z    +0.000, E1   -30.702, E3 -227353.740}
SPL {X  -155.358, Y  +344.279, Z    +0.000, E1   -24.937, E3 -227358.929}
SPL {X  -158.582, Y  +361.322, Z    +0.000, E1   -15.773, E3 -227363.272}
SPL {X  -159.657, Y  +372.183, Z    +0.000, E1    -8.995, E3 -227364.880}
SPL {X  -159.949, Y  +378.873, Z    +0.000, E1    -4.398, E3 -227365.455}
SPL {X  -159.990, Y  +382.801, Z    +0.000, E1    -1.461, E3 -227365.628}
SPL {X  -159.990, Y  +385.055, Z    +0.000, E1    +0.429, E3 -227365.668}
SPL {X  -159.990, Y  +388.743, Z    +0.000, E1    +5.147, E3 -227365.808}
SPL {X  -159.990, Y  +394.848, Z    +0.000, E1   +14.441, E3 -227366.348}
SPL {X  -159.990, Y  +402.771, Z    +0.000, E1   +27.045, E3 -227367.601}
SPL {X  -159.990, Y  +416.096, Z    +0.000, E1   +42.325, E3 -227371.268}
SPL {X  -159.990, Y  +469.763, Z    +0.000, E1   +60.937, E3 -227396.498}
SPL {X  -159.990, Y  +561.242, Z    +0.000, E1   +63.988, E3 -227467.446}
SPL {X  -159.990, Y  +574.019, Z    +0.000, E1   +64.020, E3 -227480.612}
SPL {X  -159.990, Y  +591.720, Z    +0.000, E1   +64.032, E3 -227498.911}
SPL {X  -159.990, Y  +605.088, Z    +0.000, E1   +63.988, E3 -227512.838}
SPL {X  -159.990, Y  +614.683, Z    +0.000, E1   +63.997, E3 -227522.732}
SPL {X  -159.990, Y  +629.274, Z    +0.000, E1   +64.033, E3 -227537.763}
SPL {X  -159.990, Y  +645.396, Z    +0.000, E1   +64.010, E3 -227554.495}
SPL {X  -159.990, Y  +659.675, Z    +0.000, E1   +64.013, E3 -227569.267}
SPL {X  -159.990, Y  +670.719, Z    +0.000, E1   +63.993, E3 -227580.716}
SPL {X  -159.767, Y  +679.937, Z    +0.000, E1   +63.968, E3 -227590.491}
SPL {X  -158.736, Y  +691.491, Z    +0.000, E1   +63.843, E3 -227603.490}
SPL {X  -157.131, Y  +701.612, Z    +0.000, E1   +63.591, E3 -227615.680}
SPL {X  -154.918, Y  +711.464, Z    +0.000, E1   +63.294, E3 -227628.115}
SPL {X  -151.874, Y  +721.810, Z    +0.000, E1   +62.834, E3 -227641.922}
SPL {X  -148.087, Y  +732.056, Z    +0.000, E1   +62.252, E3 -227656.278}
SPL {X  -144.667, Y  +739.825, Z    +0.000, E1   +61.658, E3 -227667.668}
SPL {X  -142.263, Y  +744.698, Z    +0.000, E1   +61.245, E3 -227674.983}
SPL {X  -139.956, Y  +749.019, Z    +0.000, E1   +60.852, E3 -227681.560}
SPL {X  -136.617, Y  +754.762, Z    +0.000, E1   +60.296, E3 -227690.415}
SPL {X  -132.995, Y  +760.433, Z    +0.000, E1   +59.601, E3 -227699.378}
SPL {X  -109.949, Y  +787.724, Z    +0.000, E1   +51.944, E3 -227791.940}
ENDSPLINE

SPLINE
SPL {X  -129.366, Y  +765.635, Z    +0.000, E1   +44.361, E3 -227901.682}
SPL {X  -144.719, Y  +739.715, Z    +0.000, E1   +37.620, E3 -227928.529}
SPL {X  -154.606, Y  +712.654, Z    +0.000, E1   +26.872, E3 -227941.749}
SPL {X  -158.229, Y  +695.175, Z    +0.000, E1   +17.621, E3 -227946.235}
SPL {X  -159.735, Y  +680.532, Z    +0.000, E1    +8.352, E3 -227948.328}
SPL {X  -159.990, Y  +671.731, Z    +0.000, E1    +1.953, E3 -227948.877}
SPL {X  -159.990, Y  +669.188, Z    +0.000, E1    -0.261, E3 -227948.922}
SPL {X  -159.990, Y  +666.135, Z    +0.000, E1    -4.178, E3 -227949.011}
SPL {X  -159.990, Y  +662.249, Z    +0.000, E1   -10.338, E3 -227949.242}
SPL {X  -159.990, Y  +658.381, Z    +0.000, E1   -16.786, E3 -227949.634}
SPL {X  -159.990, Y  +651.878, Z    +0.000, E1   -27.298, E3 -227950.633}
SPL {X  -159.990, Y  +644.587, Z    +0.000, E1   -37.284, E3 -227952.216}
SPL {X  -159.990, Y  +633.621, Z    +0.000, E1   -47.309, E3 -227955.707}
SPL {X  -159.990, Y  +588.658, Z    +0.000, E1   -60.812, E3 -227978.026}
SPL {X  -159.990, Y  +495.038, Z    +0.000, E1   -63.580, E3 -228053.263}
SPL {X  -159.990, Y  +483.848, Z    +0.000, E1   -63.590, E3 -228065.047}
SPL {X  -159.990, Y  +471.874, Z    +0.000, E1   -63.586, E3 -228077.673}
SPL {X  -159.990, Y  +461.079, Z    +0.000, E1   -63.579, E3 -228089.082}
SPL {X  -159.990, Y  +450.188, Z    +0.000, E1   -63.581, E3 -228100.572}
SPL {X  -159.990, Y  +442.553, Z    +0.000, E1   -63.337, E3 -228110.396}
ENDSPLINE

SPLINE
SPL {X  -159.990, Y  +465.419, Z    +0.000, E1   -58.181, E3 -228119.241}
ENDSPLINE

SPLINE
SPL {X  -159.990, Y  +455.003, Z    +0.000, E1   -58.788, E3 -228128.779}
SPL {X  -159.990, Y  +443.180, Z    +0.000, E1   -59.522, E3 -228138.818}
SPL {X  -159.990, Y  +431.227, Z    +0.000, E1   -60.120, E3 -228149.510}
SPL {X  -159.990, Y  +413.464, Z    +0.000, E1   -61.043, E3 -228164.500}
SPL {X  -159.990, Y  +395.417, Z    +0.000, E1   -62.063, E3 -228177.943}
SPL {X  -159.983, Y  +381.042, Z    +0.000, E1   -62.802, E3 -228188.574}
SPL {X  -159.542, Y  +370.537, Z    +0.000, E1   -63.069, E3 -228197.956}
SPL {X  -158.287, Y  +359.218, Z    +0.000, E1   -62.927, E3 -228211.371}
SPL {X  -156.553, Y  +349.515, Z    +0.000, E1   -62.627, E3 -228223.682}
SPL {X  -154.421, Y  +340.656, Z    +0.000, E1   -62.344, E3 -228235.316}
SPL {X  -151.938, Y  +332.383, Z    +0.000, E1   -61.927, E3 -228246.789}
SPL {X  -149.604, Y  +325.796, Z    +0.000, E1   -61.568, E3 -228256.175}
SPL {X  -147.413, Y  +320.320, Z    +0.000, E1   -61.198, E3 -228264.228}
SPL {X  -145.235, Y  +315.391, Z    +0.000, E1   -60.847, E3 -228271.603}
SPL {X  -142.998, Y  +310.747, Z    +0.000, E1   -60.455, E3 -228278.715}
SPL {X  -140.747, Y  +306.427, Z    +0.000, E1   -60.074, E3 -228285.424}
SPL {X  -138.010, Y  +301.568, Z    +0.000, E1   -59.585, E3 -228293.110}
SPL {X  -134.495, Y  +295.853, Z    +0.000, E1   -58.965, E3 -228302.248}
SPL {X  -113.391, Y  +269.632, Z    +0.000, E1   -50.631, E3 -228402.331}
ENDSPLINE

